LIN {X 0,Y 271.494,Z 602.071,A -85,B 0,C 180,E1 12019.317,E2 12019.317} C_VEL
LIN {X 0,Y 274.769,Z 581.052,A -85,B 0,C 180,E1 12017.936,E2 12017.936} C_VEL
LIN {X 0,Y 277.472,Z 558.924,A -85,B 0,C 180,E1 12016.896,E2 12016.896} C_VEL
LIN {X 0,Y 292.736,Z 402.476,A -85,B 0,C 180,E1 12011.469,E2 12011.469} C_VEL
LIN {X 0,Y 280.402,Z 378.491,A -85,B 0,C 180,E1 12008.156,E2 12008.156} C_VEL
LIN {X 0,Y 268.661,Z 357.396,A -85,B 0,C 180,E1 12004.711,E2 12004.711} C_VEL
LIN {X 0,Y 263.05,Z 347.539,A -85,B 0,C 180,E1 12002.855,E2 12002.855} C_VEL
LIN {X 0,Y 263.382,Z 346.943,A -85,B 0,C 180,E1 12002.565,E2 12002.565} C_VEL
LIN {X 0,Y 264.367,Z 347.015,A -85,B 0,C 180,E1 12002.274,E2 12002.274} C_VEL
LIN {X 0,Y 270.486,Z 361.582,A -85,B 0,C 180,E1 11998.605,E2 11998.605} C_VEL
LIN {X 0,Y 276.098,Z 377.318,A -85,B 0,C 180,E1 11995.128,E2 11995.128} C_VEL
LIN {X 0,Y 279.437,Z 389.009,A -85,B 0,C 180,E1 11992.846,E2 11992.846} C_VEL
LIN {X 0,Y 273.666,Z 431.774,A -85,B 0,C 180,E1 11987.985,E2 11987.985} C_VEL
LIN {X 0,Y 267.938,Z 475.725,A -85,B 0,C 180,E1 11982.94,E2 11982.94} C_VEL
LIN {X 0,Y 266.869,Z 485.441,A -85,B 0,C 180,E1 11981.853,E2 11981.853} C_VEL
LIN {X 0,Y 268.737,Z 511.468,A -85,B 0,C 180,E1 11980.723,E2 11980.723} C_VEL
LIN {X 0,Y 263.4,Z 629.84,A -85,B 0,C 180,E1 11977.527,E2 11977.527} C_VEL
LIN {X 0,Y 262.031,Z 646.203,A -85,B 0,C 180,E1 11976.686,E2 11976.686} C_VEL
LIN {X 0,Y 260.134,Z 661.581,A -85,B 0,C 180,E1 11975.516,E2 11975.516} C_VEL
LIN {X 0,Y 257.767,Z 676.09,A -85,B 0,C 180,E1 11974.006,E2 11974.006} C_VEL
LIN {X 0,Y 254.908,Z 690.584,A -85,B 0,C 180,E1 11972.025,E2 11972.025} C_VEL
LIN {X 0,Y 251.971,Z 703.426,A -85,B 0,C 180,E1 11969.752,E2 11969.752} C_VEL
LIN {X 0,Y 248.964,Z 715.561,A -85,B 0,C 180,E1 11967.01,E2 11967.01} C_VEL
LIN {X 0,Y 246.29,Z 725.681,A -85,B 0,C 180,E1 11964.066,E2 11964.066} C_VEL
LIN {X 0,Y 243.991,Z 734.43,A -85,B 0,C 180,E1 11960.806,E2 11960.806} C_VEL
LIN {X 0,Y 242.244,Z 741.402,A -85,B 0,C 180,E1 11957.367,E2 11957.367} C_VEL
LIN {X 0,Y 241.046,Z 746.913,A -85,B 0,C 180,E1 11953.619,E2 11953.619} C_VEL
LIN {X 0,Y 240.46,Z 750.406,A -85,B 0,C 180,E1 11950.01,E2 11950.01} C_VEL
LIN {X 0,Y 240.251,Z 752.346,A -85,B 0,C 180,E1 11946.194,E2 11946.194} C_VEL
LIN {X 0,Y 240.321,Z 752.618,A -85,B 0,C 180,E1 11942.401,E2 11942.401} C_VEL
LIN {X 0,Y 240.756,Z 751.048,A -85,B 0,C 180,E1 11938.451,E2 11938.451} C_VEL
LIN {X 0,Y 241.757,Z 747.721,A -85,B 0,C 180,E1 11934.565,E2 11934.565} C_VEL
LIN {X 0,Y 243.459,Z 742.459,A -85,B 0,C 180,E1 11930.772,E2 11930.772} C_VEL
LIN {X 0,Y 245.836,Z 735.559,A -85,B 0,C 180,E1 11927.222,E2 11927.222} C_VEL
LIN {X 0,Y 248.868,Z 726.664,A -85,B 0,C 180,E1 11923.842,E2 11923.842} C_VEL
LIN {X 0,Y 251.845,Z 717.662,A -85,B 0,C 180,E1 11921.176,E2 11921.176} C_VEL
LIN {X 0,Y 252.569,Z 712.778,A -85,B 0,C 180,E1 11919.813,E2 11919.813} C_VEL
LIN {X 0,Y 251.472,Z 702.77,A -85,B 0,C 180,E1 11917.085,E2 11917.085} C_VEL
LIN {X 0,Y 251.596,Z 696.374,A -85,B 0,C 180,E1 11915.677,E2 11915.677} C_VEL
LIN {X 0,Y 252.14,Z 693.786,A -85,B 0,C 180,E1 11915.218,E2 11915.218} C_VEL
LIN {X 0,Y 255.515,Z 680.254,A -85,B 0,C 180,E1 11913.284,E2 11913.284} C_VEL
LIN {X 0,Y 258.516,Z 665.707,A -85,B 0,C 180,E1 11911.697,E2 11911.697} C_VEL
LIN {X 0,Y 260.934,Z 650.294,A -85,B 0,C 180,E1 11910.46,E2 11910.46} C_VEL
LIN {X 0,Y 262.727,Z 633.392,A -85,B 0,C 180,E1 11909.54,E2 11909.54} C_VEL
LIN {X 0,Y 264.426,Z 602.955,A -85,B 0,C 180,E1 11908.631,E2 11908.631} C_VEL
LIN {X 0,Y 269.357,Z 511.316,A -85,B 0,C 180,E1 11906.141,E2 11906.141} C_VEL
LIN {X 0,Y 267.623,Z 486.252,A -85,B 0,C 180,E1 11904.737,E2 11904.737} C_VEL
LIN {X 0,Y 274.663,Z 440.447,A -85,B 0,C 180,E1 11899.475,E2 11899.475} C_VEL
LIN {X 0,Y 281.678,Z 396.905,A -85,B 0,C 180,E1 11894.519,E2 11894.519} C_VEL
LIN {X 0,Y 278.503,Z 384.661,A -85,B 0,C 180,E1 11891.599,E2 11891.599} C_VEL
LIN {X 0,Y 275.112,Z 374.138,A -85,B 0,C 180,E1 11888.57,E2 11888.57} C_VEL
LIN {X 0,Y 271.329,Z 364.565,A -85,B 0,C 180,E1 11885.287,E2 11885.287} C_VEL
LIN {X 0,Y 268.101,Z 357.243,A -85,B 0,C 180,E1 11882.138,E2 11882.138} C_VEL
LIN {X 0,Y 265.809,Z 352.672,A -85,B 0,C 180,E1 11879.785,E2 11879.785} C_VEL
LIN {X 0,Y 264.137,Z 348.957,A -85,B 0,C 180,E1 11877.614,E2 11877.614} C_VEL
LIN {X 0,Y 262.032,Z 344.964,A -85,B 0,C 180,E1 11874.746,E2 11874.746} C_VEL
LIN {X 0,Y 261.21,Z 343.736,A -85,B 0,C 180,E1 11873.407,E2 11873.407} C_VEL
LIN {X 0,Y 259.249,Z 339.266,A -85,B 0,C 180,E1 11868.395,E2 11868.395} C_VEL
LIN {X 0,Y 258.446,Z 338.509,A -85,B 0,C 180,E1 11862.437,E2 11862.437} C_VEL
LIN {X 0,Y 259.489,Z 339.421,A -85,B 0,C 180,E1 11858.053,E2 11858.053} C_VEL
LIN {X 0,Y 259.379,Z 345.514,A -85,B 0,C 180,E1 11855.155,E2 11855.155} C_VEL
LIN {X 0,Y 259.573,Z 350.003,A -85,B 0,C 180,E1 11853.615,E2 11853.615} C_VEL
LIN {X 0,Y 271.338,Z 369.415,A -85,B 0,C 180,E1 11849.925,E2 11849.925} C_VEL
LIN {X 0,Y 283.805,Z 391.256,A -85,B 0,C 180,E1 11846.389,E2 11846.389} C_VEL
LIN {X 0,Y 291.694,Z 406.109,A -85,B 0,C 180,E1 11844.305,E2 11844.305} C_VEL
LIN {X 0,Y 274.876,Z 575.506,A -85,B 0,C 180,E1 11838.587,E2 11838.587} C_VEL
LIN {X 0,Y 271.832,Z 596.932,A -85,B 0,C 180,E1 11837.513,E2 11837.513} C_VEL
LIN {X 0,Y 268.025,Z 618.404,A -85,B 0,C 180,E1 11836.049,E2 11836.049} C_VEL
LIN {X 0,Y 263.729,Z 638.906,A -85,B 0,C 180,E1 11834.23,E2 11834.23} C_VEL
LIN {X 0,Y 259.299,Z 657.672,A -85,B 0,C 180,E1 11832.136,E2 11832.136} C_VEL
LIN {X 0,Y 254.654,Z 675.677,A -85,B 0,C 180,E1 11829.656,E2 11829.656} C_VEL
LIN {X 0,Y 249.995,Z 692.7,A -85,B 0,C 180,E1 11826.779,E2 11826.779} C_VEL
LIN {X 0,Y 245.488,Z 708.606,A -85,B 0,C 180,E1 11823.493,E2 11823.493} C_VEL
LIN {X 0,Y 241.388,Z 723.196,A -85,B 0,C 180,E1 11819.802,E2 11819.802} C_VEL
LIN {X 0,Y 238.102,Z 736.125,A -85,B 0,C 180,E1 11816.021,E2 11816.021} C_VEL
LIN {X 0,Y 235.984,Z 746.974,A -85,B 0,C 180,E1 11812.676,E2 11812.676} C_VEL
LIN {X 0,Y 234.301,Z 755.943,A -85,B 0,C 180,E1 11809.18,E2 11809.18} C_VEL
LIN {X 0,Y 233.077,Z 763.404,A -85,B 0,C 180,E1 11805.422,E2 11805.422} C_VEL
LIN {X 0,Y 232.378,Z 769.258,A -85,B 0,C 180,E1 11801.413,E2 11801.413} C_VEL
LIN {X 0,Y 232.172,Z 772.992,A -85,B 0,C 180,E1 11797.669,E2 11797.669} C_VEL
LIN {X 0,Y 232.21,Z 775.067,A -85,B 0,C 180,E1 11793.948,E2 11793.948} C_VEL
LIN {X 0,Y 232.292,Z 775.579,A -85,B 0,C 180,E1 11790.244,E2 11790.244} C_VEL
LIN {X 0,Y 232.233,Z 775.277,A -85,B 0,C 180,E1 11787.036,E2 11787.036} C_VEL
LIN {X 0,Y 232.091,Z 774.894,A -85,B 0,C 180,E1 11782.82,E2 11782.82} C_VEL
LIN {X 0,Y 232.348,Z 773.008,A -85,B 0,C 180,E1 11778.077,E2 11778.077} C_VEL
LIN {X 0,Y 233.577,Z 769.389,A -85,B 0,C 180,E1 11773.075,E2 11773.075} C_VEL
LIN {X 0,Y 236.446,Z 763.468,A -85,B 0,C 180,E1 11767.628,E2 11767.628} C_VEL
LIN {X 0,Y 241.157,Z 755.58,A -85,B 0,C 180,E1 11762.329,E2 11762.329} C_VEL
LIN {X 0,Y 248.196,Z 745.291,A -85,B 0,C 180,E1 11757.051,E2 11757.051} C_VEL
LIN {X 0,Y 257.447,Z 732.968,A -85,B 0,C 180,E1 11752.145,E2 11752.145} C_VEL
LIN {X 0,Y 269.502,Z 718.104,A -85,B 0,C 180,E1 11747.526,E2 11747.526} C_VEL
LIN {X 0,Y 283.352,Z 702.222,A -85,B 0,C 180,E1 11743.663,E2 11743.663} C_VEL
LIN {X 0,Y 289.035,Z 696.015,A -85,B 0,C 180,E1 11742.353,E2 11742.353} C_VEL
LIN {X 0,Y 275.346,Z 709.401,A -85,B 0,C 180,E1 11738.917,E2 11738.917} C_VEL
LIN {X 0,Y 263.037,Z 721.802,A -85,B 0,C 180,E1 11734.762,E2 11734.762} C_VEL
LIN {X 0,Y 252.946,Z 732.321,A -85,B 0,C 180,E1 11730.132,E2 11730.132} C_VEL
LIN {X 0,Y 245.312,Z 740.47,A -85,B 0,C 180,E1 11725.338,E2 11725.338} C_VEL
LIN {X 0,Y 239.818,Z 746.395,A -85,B 0,C 180,E1 11720.5,E2 11720.5} C_VEL
LIN {X 0,Y 236.002,Z 750.456,A -85,B 0,C 180,E1 11715.48,E2 11715.48} C_VEL
LIN {X 0,Y 233.765,Z 752.545,A -85,B 0,C 180,E1 11710.597,E2 11710.597} C_VEL
LIN {X 0,Y 232.675,Z 752.869,A -85,B 0,C 180,E1 11705.919,E2 11705.919} C_VEL
LIN {X 0,Y 232.274,Z 751.624,A -85,B 0,C 180,E1 11701.479,E2 11701.479} C_VEL
LIN {X 0,Y 232.176,Z 749.013,A -85,B 0,C 180,E1 11697.284,E2 11697.284} C_VEL
LIN {X 0,Y 232.325,Z 744.909,A -85,B 0,C 180,E1 11693.078,E2 11693.078} C_VEL
LIN {X 0,Y 232.887,Z 739.168,A -85,B 0,C 180,E1 11688.859,E2 11688.859} C_VEL
LIN {X 0,Y 234.051,Z 731.644,A -85,B 0,C 180,E1 11684.64,E2 11684.64} C_VEL
LIN {X 0,Y 235.982,Z 722.115,A -85,B 0,C 180,E1 11680.443,E2 11680.443} C_VEL
LIN {X 0,Y 238.593,Z 711.091,A -85,B 0,C 180,E1 11676.539,E2 11676.539} C_VEL
LIN {X 0,Y 241.789,Z 698.652,A -85,B 0,C 180,E1 11672.942,E2 11672.942} C_VEL
LIN {X 0,Y 245.586,Z 684.276,A -85,B 0,C 180,E1 11669.543,E2 11669.543} C_VEL
LIN {X 0,Y 249.754,Z 668.328,A -85,B 0,C 180,E1 11666.463,E2 11666.463} C_VEL
LIN {X 0,Y 254.158,Z 650.692,A -85,B 0,C 180,E1 11663.695,E2 11663.695} C_VEL
LIN {X 0,Y 258.477,Z 632.032,A -85,B 0,C 180,E1 11661.337,E2 11661.337} C_VEL
LIN {X 0,Y 262.541,Z 612.369,A -85,B 0,C 180,E1 11659.364,E2 11659.364} C_VEL
LIN {X 0,Y 266.041,Z 592.568,A -85,B 0,C 180,E1 11657.821,E2 11657.821} C_VEL
LIN {X 0,Y 269.162,Z 571.164,A -85,B 0,C 180,E1 11656.579,E2 11656.579} C_VEL
LIN {X 0,Y 272.248,Z 542.164,A -85,B 0,C 180,E1 11655.408,E2 11655.408} C_VEL
LIN {X 0,Y 286.213,Z 405.215,A -85,B 0,C 180,E1 11650.561,E2 11650.561} C_VEL
LIN {X 0,Y 274.152,Z 381.732,A -85,B 0,C 180,E1 11647.196,E2 11647.196} C_VEL
LIN {X 0,Y 263.313,Z 362.162,A -85,B 0,C 180,E1 11643.9,E2 11643.9} C_VEL
LIN {X 0,Y 259.462,Z 355.12,A -85,B 0,C 180,E1 11642.544,E2 11642.544} C_VEL
LIN {X 0,Y 259.948,Z 354.608,A -85,B 0,C 180,E1 11642.197,E2 11642.197} C_VEL
LIN {X 0,Y 265.947,Z 369.757,A -85,B 0,C 180,E1 11638.386,E2 11638.386} C_VEL
LIN {X 0,Y 270.932,Z 384.639,A -85,B 0,C 180,E1 11635.115,E2 11635.115} C_VEL
LIN {X 0,Y 272.965,Z 392.002,A -85,B 0,C 180,E1 11633.66,E2 11633.66} C_VEL
LIN {X 0,Y 267.1,Z 433.334,A -85,B 0,C 180,E1 11628.895,E2 11628.895} C_VEL
LIN {X 0,Y 261.43,Z 474.987,A -85,B 0,C 180,E1 11624.058,E2 11624.058} C_VEL
LIN {X 0,Y 260.198,Z 485.826,A -85,B 0,C 180,E1 11622.836,E2 11622.836} C_VEL
LIN {X 0,Y 262.029,Z 512.287,A -85,B 0,C 180,E1 11621.656,E2 11621.656} C_VEL
LIN {X 0,Y 256.451,Z 630.322,A -85,B 0,C 180,E1 11618.395,E2 11618.395} C_VEL
LIN {X 0,Y 255.011,Z 646.741,A -85,B 0,C 180,E1 11617.529,E2 11617.529} C_VEL
LIN {X 0,Y 253.07,Z 661.849,A -85,B 0,C 180,E1 11616.354,E2 11616.354} C_VEL
LIN {X 0,Y 250.605,Z 676.391,A -85,B 0,C 180,E1 11614.809,E2 11614.809} C_VEL
LIN {X 0,Y 247.624,Z 690.905,A -85,B 0,C 180,E1 11612.78,E2 11612.78} C_VEL
LIN {X 0,Y 244.589,Z 703.65,A -85,B 0,C 180,E1 11610.471,E2 11610.471} C_VEL
LIN {X 0,Y 241.413,Z 715.913,A -85,B 0,C 180,E1 11607.629,E2 11607.629} C_VEL
LIN {X 0,Y 238.505,Z 726.419,A -85,B 0,C 180,E1 11604.47,E2 11604.47} C_VEL
LIN {X 0,Y 236.196,Z 734.801,A -85,B 0,C 180,E1 11601.237,E2 11601.237} C_VEL
LIN {X 0,Y 234.356,Z 741.78,A -85,B 0,C 180,E1 11597.686,E2 11597.686} C_VEL
LIN {X 0,Y 233.093,Z 747.297,A -85,B 0,C 180,E1 11593.813,E2 11593.813} C_VEL
LIN {X 0,Y 232.482,Z 750.755,A -85,B 0,C 180,E1 11590.141,E2 11590.141} C_VEL
LIN {X 0,Y 232.258,Z 752.739,A -85,B 0,C 180,E1 11586.133,E2 11586.133} C_VEL
LIN {X 0,Y 232.336,Z 753.025,A -85,B 0,C 180,E1 11582.308,E2 11582.308} C_VEL
LIN {X 0,Y 232.802,Z 751.526,A -85,B 0,C 180,E1 11578.256,E2 11578.256} C_VEL
LIN {X 0,Y 233.903,Z 748.174,A -85,B 0,C 180,E1 11574.156,E2 11574.156} C_VEL
LIN {X 0,Y 235.607,Z 743.314,A -85,B 0,C 180,E1 11570.468,E2 11570.468} C_VEL
LIN {X 0,Y 238.092,Z 736.561,A -85,B 0,C 180,E1 11566.807,E2 11566.807} C_VEL
LIN {X 0,Y 241.11,Z 728.302,A -85,B 0,C 180,E1 11563.477,E2 11563.477} C_VEL
LIN {X 0,Y 244.661,Z 718.184,A -85,B 0,C 180,E1 11560.353,E2 11560.353} C_VEL
LIN {X 0,Y 248.154,Z 707.442,A -85,B 0,C 180,E1 11557.767,E2 11557.767} C_VEL
LIN {X 0,Y 251.913,Z 694.598,A -85,B 0,C 180,E1 11555.355,E2 11555.355} C_VEL
LIN {X 0,Y 252.14,Z 693.786,A -85,B 0,C 180,E1 11555.218,E2 11555.218} C_VEL
LIN {X 0,Y 252.943,Z 687.681,A -85,B 0,C 180,E1 11554.142,E2 11554.142} C_VEL
LIN {X 0,Y 251.846,Z 673.719,A -85,B 0,C 180,E1 11551.616,E2 11551.616} C_VEL
LIN {X 0,Y 252.061,Z 667.063,A -85,B 0,C 180,E1 11550.711,E2 11550.711} C_VEL
LIN {X 0,Y 252.375,Z 665.07,A -85,B 0,C 180,E1 11550.503,E2 11550.503} C_VEL
LIN {X 0,Y 254.891,Z 649.347,A -85,B 0,C 180,E1 11549.257,E2 11549.257} C_VEL
LIN {X 0,Y 256.677,Z 632.86,A -85,B 0,C 180,E1 11548.369,E2 11548.369} C_VEL
LIN {X 0,Y 260.151,Z 572.276,A -85,B 0,C 180,E1 11546.628,E2 11546.628} C_VEL
LIN {X 0,Y 263.538,Z 512.271,A -85,B 0,C 180,E1 11544.968,E2 11544.968} C_VEL
LIN {X 0,Y 261.859,Z 487.034,A -85,B 0,C 180,E1 11543.517,E2 11543.517} C_VEL
LIN {X 0,Y 269.118,Z 441.982,A -85,B 0,C 180,E1 11538.298,E2 11538.298} C_VEL
LIN {X 0,Y 276.117,Z 400.724,A -85,B 0,C 180,E1 11533.561,E2 11533.561} C_VEL
LIN {X 0,Y 273.39,Z 389.42,A -85,B 0,C 180,E1 11530.751,E2 11530.751} C_VEL
LIN {X 0,Y 270.594,Z 380.2,A -85,B 0,C 180,E1 11528.02,E2 11528.02} C_VEL
LIN {X 0,Y 267.148,Z 370.865,A -85,B 0,C 180,E1 11524.724,E2 11524.724} C_VEL
LIN {X 0,Y 264.039,Z 363.618,A -85,B 0,C 180,E1 11521.52,E2 11521.52} C_VEL
LIN {X 0,Y 262.156,Z 359.505,A -85,B 0,C 180,E1 11519.345,E2 11519.345} C_VEL
LIN {X 0,Y 260.523,Z 355.857,A -85,B 0,C 180,E1 11517.141,E2 11517.141} C_VEL
LIN {X 0,Y 258.425,Z 351.439,A -85,B 0,C 180,E1 11513.782,E2 11513.782} C_VEL
LIN {X 0,Y 256.516,Z 347.354,A -85,B 0,C 180,E1 11509.173,E2 11509.173} C_VEL
LIN {X 0,Y 256.252,Z 346.625,A -85,B 0,C 180,E1 11507.837,E2 11507.837} C_VEL
LIN {X 0,Y 255.772,Z 346.054,A -85,B 0,C 180,E1 11502.248,E2 11502.248} C_VEL
LIN {X 0,Y 256.678,Z 346.655,A -85,B 0,C 180,E1 11498.521,E2 11498.521} C_VEL
LIN {X 0,Y 256.428,Z 352.391,A -85,B 0,C 180,E1 11495.833,E2 11495.833} C_VEL
LIN {X 0,Y 256.52,Z 358.28,A -85,B 0,C 180,E1 11493.775,E2 11493.775} C_VEL
LIN {X 0,Y 268.181,Z 377.95,A -85,B 0,C 180,E1 11490.059,E2 11490.059} C_VEL
LIN {X 0,Y 280.331,Z 399.558,A -85,B 0,C 180,E1 11486.573,E2 11486.573} C_VEL
LIN {X 0,Y 285.231,Z 409.114,A -85,B 0,C 180,E1 11485.228,E2 11485.228} C_VEL
LIN {X 0,Y 268.013,Z 575.619,A -85,B 0,C 180,E1 11479.454,E2 11479.454} C_VEL
LIN {X 0,Y 264.884,Z 596.863,A -85,B 0,C 180,E1 11478.36,E2 11478.36} C_VEL
LIN {X 0,Y 260.978,Z 618.204,A -85,B 0,C 180,E1 11476.869,E2 11476.869} C_VEL
LIN {X 0,Y 256.566,Z 638.64,A -85,B 0,C 180,E1 11475.013,E2 11475.013} C_VEL
LIN {X 0,Y 251.791,Z 658.206,A -85,B 0,C 180,E1 11472.765,E2 11472.765} C_VEL
LIN {X 0,Y 247.008,Z 676.133,A -85,B 0,C 180,E1 11470.209,E2 11470.209} C_VEL
LIN {X 0,Y 242.353,Z 692.634,A -85,B 0,C 180,E1 11467.331,E2 11467.331} C_VEL
LIN {X 0,Y 237.684,Z 708.623,A -85,B 0,C 180,E1 11463.918,E2 11463.918} C_VEL
LIN {X 0,Y 233.255,Z 724.496,A -85,B 0,C 180,E1 11459.889,E2 11459.889} C_VEL
LIN {X 0,Y 230.681,Z 736.731,A -85,B 0,C 180,E1 11456.764,E2 11456.764} C_VEL
LIN {X 0,Y 228.298,Z 747.641,A -85,B 0,C 180,E1 11453.211,E2 11453.211} C_VEL
LIN {X 0,Y 226.476,Z 756.403,A -85,B 0,C 180,E1 11449.601,E2 11449.601} C_VEL
LIN {X 0,Y 225.149,Z 763.621,A -85,B 0,C 180,E1 11445.714,E2 11445.714} C_VEL
LIN {X 0,Y 224.392,Z 769.313,A -85,B 0,C 180,E1 11441.564,E2 11441.564} C_VEL
LIN {X 0,Y 224.168,Z 773.013,A -85,B 0,C 180,E1 11437.429,E2 11437.429} C_VEL
LIN {X 0,Y 224.224,Z 774.858,A -85,B 0,C 180,E1 11433.576,E2 11433.576} C_VEL
LIN {X 0,Y 224.304,Z 775.142,A -85,B 0,C 180,E1 11429.742,E2 11429.742} C_VEL
LIN {X 0,Y 224.239,Z 774.681,A -85,B 0,C 180,E1 11426.674,E2 11426.674} C_VEL
LIN {X 0,Y 224.104,Z 774.334,A -85,B 0,C 180,E1 11422.047,E2 11422.047} C_VEL
LIN {X 0,Y 224.526,Z 772.338,A -85,B 0,C 180,E1 11416.87,E2 11416.87} C_VEL
LIN {X 0,Y 226.218,Z 768.472,A -85,B 0,C 180,E1 11411.441,E2 11411.441} C_VEL
LIN {X 0,Y 229.7,Z 762.535,A -85,B 0,C 180,E1 11405.845,E2 11405.845} C_VEL
LIN {X 0,Y 235.455,Z 754.321,A -85,B 0,C 180,E1 11400.206,E2 11400.206} C_VEL
LIN {X 0,Y 243.487,Z 744.149,A -85,B 0,C 180,E1 11394.905,E2 11394.905} C_VEL
LIN {X 0,Y 254.295,Z 731.59,A -85,B 0,C 180,E1 11389.845,E2 11389.845} C_VEL
LIN {X 0,Y 267.584,Z 717.288,A -85,B 0,C 180,E1 11385.371,E2 11385.371} C_VEL
LIN {X 0,Y 279.674,Z 705.089,A -85,B 0,C 180,E1 11382.299,E2 11382.299} C_VEL
LIN {X 0,Y 265.174,Z 717.754,A -85,B 0,C 180,E1 11378.472,E2 11378.472} C_VEL
LIN {X 0,Y 252.612,Z 729.11,A -85,B 0,C 180,E1 11373.923,E2 11373.923} C_VEL
LIN {X 0,Y 242.853,Z 738.169,A -85,B 0,C 180,E1 11369.066,E2 11369.066} C_VEL
LIN {X 0,Y 235.58,Z 744.978,A -85,B 0,C 180,E1 11364.044,E2 11364.044} C_VEL
LIN {X 0,Y 230.269,Z 749.837,A -85,B 0,C 180,E1 11358.742,E2 11358.742} C_VEL
LIN {X 0,Y 226.95,Z 752.62,A -85,B 0,C 180,E1 11353.502,E2 11353.502} C_VEL
LIN {X 0,Y 225.16,Z 753.534,A -85,B 0,C 180,E1 11348.426,E2 11348.426} C_VEL
LIN {X 0,Y 224.408,Z 752.743,A -85,B 0,C 180,E1 11343.553,E2 11343.553} C_VEL
LIN {X 0,Y 224.198,Z 750.439,A -85,B 0,C 180,E1 11338.977,E2 11338.977} C_VEL
LIN {X 0,Y 224.234,Z 746.715,A -85,B 0,C 180,E1 11334.626,E2 11334.626} C_VEL
LIN {X 0,Y 224.634,Z 741.414,A -85,B 0,C 180,E1 11330.261,E2 11330.261} C_VEL
LIN {X 0,Y 225.605,Z 734.39,A -85,B 0,C 180,E1 11325.891,E2 11325.891} C_VEL
LIN {X 0,Y 227.332,Z 725.447,A -85,B 0,C 180,E1 11321.537,E2 11321.537} C_VEL
LIN {X 0,Y 229.76,Z 715.051,A -85,B 0,C 180,E1 11317.482,E2 11317.482} C_VEL
LIN {X 0,Y 232.803,Z 703.296,A -85,B 0,C 180,E1 11313.744,E2 11313.744} C_VEL
LIN {X 0,Y 236.612,Z 689.242,A -85,B 0,C 180,E1 11310.089,E2 11310.089} C_VEL
LIN {X 0,Y 240.871,Z 673.589,A -85,B 0,C 180,E1 11306.773,E2 11306.773} C_VEL
LIN {X 0,Y 245.425,Z 656.201,A -85,B 0,C 180,E1 11303.79,E2 11303.79} C_VEL
LIN {X 0,Y 249.925,Z 637.749,A -85,B 0,C 180,E1 11301.251,E2 11301.251} C_VEL
LIN {X 0,Y 254.246,Z 618.089,A -85,B 0,C 180,E1 11299.095,E2 11299.095} C_VEL
LIN {X 0,Y 258.195,Z 597.49,A -85,B 0,C 180,E1 11297.336,E2 11297.336} C_VEL
LIN {X 0,Y 261.59,Z 576.13,A -85,B 0,C 180,E1 11295.958,E2 11295.958} C_VEL
LIN {X 0,Y 264.306,Z 553.841,A -85,B 0,C 180,E1 11294.945,E2 11294.945} C_VEL
LIN {X 0,Y 279.796,Z 408.146,A -85,B 0,C 180,E1 11289.649,E2 11289.649} C_VEL
LIN {X 0,Y 267.51,Z 384.104,A -85,B 0,C 180,E1 11286.066,E2 11286.066} C_VEL
LIN {X 0,Y 256.178,Z 363.663,A -85,B 0,C 180,E1 11282.459,E2 11282.459} C_VEL
LIN {X 0,Y 255.776,Z 362.628,A -85,B 0,C 180,E1 11282.119,E2 11282.119} C_VEL
LIN {X 0,Y 256.512,Z 364.958,A -85,B 0,C 180,E1 11281.388,E2 11281.388} C_VEL
LIN {X 0,Y 262.035,Z 379.972,A -85,B 0,C 180,E1 11277.715,E2 11277.715} C_VEL
LIN {X 0,Y 266.545,Z 394.897,A -85,B 0,C 180,E1 11274.52,E2 11274.52} C_VEL
LIN {X 0,Y 260.248,Z 437.782,A -85,B 0,C 180,E1 11269.529,E2 11269.529} C_VEL
LIN {X 0,Y 254.152,Z 480.628,A -85,B 0,C 180,E1 11264.469,E2 11264.469} C_VEL
LIN {X 0,Y 253.586,Z 486.33,A -85,B 0,C 180,E1 11263.854,E2 11263.854} C_VEL
LIN {X 0,Y 255.345,Z 513.166,A -85,B 0,C 180,E1 11262.622,E2 11262.622} C_VEL
LIN {X 0,Y 249.556,Z 630.626,A -85,B 0,C 180,E1 11259.312,E2 11259.312} C_VEL
LIN {X 0,Y 248.068,Z 646.977,A -85,B 0,C 180,E1 11258.433,E2 11258.433} C_VEL
LIN {X 0,Y 246.058,Z 662.048,A -85,B 0,C 180,E1 11257.239,E2 11257.239} C_VEL
LIN {X 0,Y 243.492,Z 676.649,A -85,B 0,C 180,E1 11255.658,E2 11255.658} C_VEL
LIN {X 0,Y 240.384,Z 691.194,A -85,B 0,C 180,E1 11253.58,E2 11253.58} C_VEL
LIN {X 0,Y 237.215,Z 703.971,A -85,B 0,C 180,E1 11251.21,E2 11251.21} C_VEL
LIN {X 0,Y 233.891,Z 716.252,A -85,B 0,C 180,E1 11248.288,E2 11248.288} C_VEL
LIN {X 0,Y 231.057,Z 726.056,A -85,B 0,C 180,E1 11245.287,E2 11245.287} C_VEL
LIN {X 0,Y 228.39,Z 735.262,A -85,B 0,C 180,E1 11241.657,E2 11241.657} C_VEL
LIN {X 0,Y 226.476,Z 742.158,A -85,B 0,C 180,E1 11238.027,E2 11238.027} C_VEL
LIN {X 0,Y 225.141,Z 747.679,A -85,B 0,C 180,E1 11234.021,E2 11234.021} C_VEL
LIN {X 0,Y 224.477,Z 751.264,A -85,B 0,C 180,E1 11230.027,E2 11230.027} C_VEL
LIN {X 0,Y 224.265,Z 753.211,A -85,B 0,C 180,E1 11225.788,E2 11225.788} C_VEL
LIN {X 0,Y 224.38,Z 753.375,A -85,B 0,C 180,E1 11221.817,E2 11221.817} C_VEL
LIN {X 0,Y 224.933,Z 751.769,A -85,B 0,C 180,E1 11217.629,E2 11217.629} C_VEL
LIN {X 0,Y 226.112,Z 748.514,A -85,B 0,C 180,E1 11213.593,E2 11213.593} C_VEL
LIN {X 0,Y 228.106,Z 743.271,A -85,B 0,C 180,E1 11209.558,E2 11209.558} C_VEL
LIN {X 0,Y 230.839,Z 736.383,A -85,B 0,C 180,E1 11205.789,E2 11205.789} C_VEL
LIN {X 0,Y 234.113,Z 727.94,A -85,B 0,C 180,E1 11202.371,E2 11202.371} C_VEL
LIN {X 0,Y 237.761,Z 718.16,A -85,B 0,C 180,E1 11199.311,E2 11199.311} C_VEL
LIN {X 0,Y 241.601,Z 706.878,A -85,B 0,C 180,E1 11196.581,E2 11196.581} C_VEL
LIN {X 0,Y 245.637,Z 693.669,A -85,B 0,C 180,E1 11194.098,E2 11194.098} C_VEL
LIN {X 0,Y 249.157,Z 680.091,A -85,B 0,C 180,E1 11192.147,E2 11192.147} C_VEL
LIN {X 0,Y 252.375,Z 665.07,A -85,B 0,C 180,E1 11190.503,E2 11190.503} C_VEL
LIN {X 0,Y 252.892,Z 658.091,A -85,B 0,C 180,E1 11189.73,E2 11189.73} C_VEL
LIN {X 0,Y 251.256,Z 644.385,A -85,B 0,C 180,E1 11188.045,E2 11188.045} C_VEL
LIN {X 0,Y 250.603,Z 636.11,A -85,B 0,C 180,E1 11187.324,E2 11187.324} C_VEL
LIN {X 0,Y 250.705,Z 632.868,A -85,B 0,C 180,E1 11187.162,E2 11187.162} C_VEL
LIN {X 0,Y 257.896,Z 513.32,A -85,B 0,C 180,E1 11183.734,E2 11183.734} C_VEL
LIN {X 0,Y 256.313,Z 487.239,A -85,B 0,C 180,E1 11182.175,E2 11182.175} C_VEL
LIN {X 0,Y 264.093,Z 441.625,A -85,B 0,C 180,E1 11176.837,E2 11176.837} C_VEL
LIN {X 0,Y 270.737,Z 404.278,A -85,B 0,C 180,E1 11172.478,E2 11172.478} C_VEL
LIN {X 0,Y 268.321,Z 393.587,A -85,B 0,C 180,E1 11169.654,E2 11169.654} C_VEL
LIN {X 0,Y 265.327,Z 384.015,A -85,B 0,C 180,E1 11166.709,E2 11166.709} C_VEL
LIN {X 0,Y 262.014,Z 374.57,A -85,B 0,C 180,E1 11163.063,E2 11163.063} C_VEL
LIN {X 0,Y 258.867,Z 366.992,A -85,B 0,C 180,E1 11159.337,E2 11159.337} C_VEL
LIN {X 0,Y 256.999,Z 362.781,A -85,B 0,C 180,E1 11156.655,E2 11156.655} C_VEL
LIN {X 0,Y 255.254,Z 358.691,A -85,B 0,C 180,E1 11153.478,E2 11153.478} C_VEL
LIN {X 0,Y 253.568,Z 354.666,A -85,B 0,C 180,E1 11148.86,E2 11148.86} C_VEL
LIN {X 0,Y 253.229,Z 353.955,A -85,B 0,C 180,E1 11147.215,E2 11147.215} C_VEL
LIN {X 0,Y 253.131,Z 353.618,A -85,B 0,C 180,E1 11141.58,E2 11141.58} C_VEL
LIN {X 0,Y 253.853,Z 354.345,A -85,B 0,C 180,E1 11138.755,E2 11138.755} C_VEL
LIN {X 0,Y 253.469,Z 359.89,A -85,B 0,C 180,E1 11136.275,E2 11136.275} C_VEL
LIN {X 0,Y 253.446,Z 366.618,A -85,B 0,C 180,E1 11133.936,E2 11133.936} C_VEL
LIN {X 0,Y 265.525,Z 387.341,A -85,B 0,C 180,E1 11130.04,E2 11130.04} C_VEL
LIN {X 0,Y 278.506,Z 411.075,A -85,B 0,C 180,E1 11126.282,E2 11126.282} C_VEL
LIN {X 0,Y 278.766,Z 412.273,A -85,B 0,C 180,E1 11126.173,E2 11126.173} C_VEL
LIN {X 0,Y 261.181,Z 575.534,A -85,B 0,C 180,E1 11120.356,E2 11120.356} C_VEL
LIN {X 0,Y 257.863,Z 597.286,A -85,B 0,C 180,E1 11119.203,E2 11119.203} C_VEL
LIN {X 0,Y 253.989,Z 617.808,A -85,B 0,C 180,E1 11117.734,E2 11117.734} C_VEL
LIN {X 0,Y 249.454,Z 638.208,A -85,B 0,C 180,E1 11115.841,E2 11115.841} C_VEL
LIN {X 0,Y 244.562,Z 657.679,A -85,B 0,C 180,E1 11113.554,E2 11113.554} C_VEL
LIN {X 0,Y 239.614,Z 675.697,A -85,B 0,C 180,E1 11110.925,E2 11110.925} C_VEL
LIN {X 0,Y 234.634,Z 692.797,A -85,B 0,C 180,E1 11107.849,E2 11107.849} C_VEL
LIN {X 0,Y 229.682,Z 709.307,A -85,B 0,C 180,E1 11104.198,E2 11104.198} C_VEL
LIN {X 0,Y 226.058,Z 725.598,A -85,B 0,C 180,E1 11100.717,E2 11100.717} C_VEL
LIN {X 0,Y 223.452,Z 736.747,A -85,B 0,C 180,E1 11097.73,E2 11097.73} C_VEL
LIN {X 0,Y 220.803,Z 747.635,A -85,B 0,C 180,E1 11094.047,E2 11094.047} C_VEL
LIN {X 0,Y 218.785,Z 756.288,A -85,B 0,C 180,E1 11090.32,E2 11090.32} C_VEL
LIN {X 0,Y 217.227,Z 763.841,A -85,B 0,C 180,E1 11086.029,E2 11086.029} C_VEL
LIN {X 0,Y 216.438,Z 769.056,A -85,B 0,C 180,E1 11081.995,E2 11081.995} C_VEL
LIN {X 0,Y 216.175,Z 772.697,A -85,B 0,C 180,E1 11077.705,E2 11077.705} C_VEL
LIN {X 0,Y 216.227,Z 774.497,A -85,B 0,C 180,E1 11073.709,E2 11073.709} C_VEL
LIN {X 0,Y 216.314,Z 774.74,A -85,B 0,C 180,E1 11069.732,E2 11069.732} C_VEL
LIN {X 0,Y 216.248,Z 774.064,A -85,B 0,C 180,E1 11066.286,E2 11066.286} C_VEL
LIN {X 0,Y 216.12,Z 773.83,A -85,B 0,C 180,E1 11061.484,E2 11061.484} C_VEL
LIN {X 0,Y 216.608,Z 772.136,A -85,B 0,C 180,E1 11056.381,E2 11056.381} C_VEL
LIN {X 0,Y 218.617,Z 768.29,A -85,B 0,C 180,E1 11050.493,E2 11050.493} C_VEL
LIN {X 0,Y 222.507,Z 762.588,A -85,B 0,C 180,E1 11044.727,E2 11044.727} C_VEL
LIN {X 0,Y 228.901,Z 754.64,A -85,B 0,C 180,E1 11038.885,E2 11038.885} C_VEL
LIN {X 0,Y 237.898,Z 744.644,A -85,B 0,C 180,E1 11033.355,E2 11033.355} C_VEL
LIN {X 0,Y 249.536,Z 732.752,A -85,B 0,C 180,E1 11028.304,E2 11028.304} C_VEL
LIN {X 0,Y 264.301,Z 718.748,A -85,B 0,C 180,E1 11023.731,E2 11023.731} C_VEL
LIN {X 0,Y 270.243,Z 713.321,A -85,B 0,C 180,E1 11022.269,E2 11022.269} C_VEL
LIN {X 0,Y 254.966,Z 725.279,A -85,B 0,C 180,E1 11018.001,E2 11018.001} C_VEL
LIN {X 0,Y 242.522,Z 735.299,A -85,B 0,C 180,E1 11013.18,E2 11013.18} C_VEL
LIN {X 0,Y 233.128,Z 742.927,A -85,B 0,C 180,E1 11008.149,E2 11008.149} C_VEL
LIN {X 0,Y 226.145,Z 748.507,A -85,B 0,C 180,E1 11002.896,E2 11002.896} C_VEL
LIN {X 0,Y 221.197,Z 752.221,A -85,B 0,C 180,E1 10997.357,E2 10997.357} C_VEL
LIN {X 0,Y 218.355,Z 753.923,A -85,B 0,C 180,E1 10992.159,E2 10992.159} C_VEL
LIN {X 0,Y 216.847,Z 753.922,A -85,B 0,C 180,E1 10986.884,E2 10986.884} C_VEL
LIN {X 0,Y 216.309,Z 752.398,A -85,B 0,C 180,E1 10982.118,E2 10982.118} C_VEL
LIN {X 0,Y 216.179,Z 749.422,A -85,B 0,C 180,E1 10977.527,E2 10977.527} C_VEL
LIN {X 0,Y 216.321,Z 745.098,A -85,B 0,C 180,E1 10973.097,E2 10973.097} C_VEL
LIN {X 0,Y 216.981,Z 738.666,A -85,B 0,C 180,E1 10968.301,E2 10968.301} C_VEL
LIN {X 0,Y 218.301,Z 730.723,A -85,B 0,C 180,E1 10963.775,E2 10963.775} C_VEL
LIN {X 0,Y 220.483,Z 720.753,A -85,B 0,C 180,E1 10959.284,E2 10959.284} C_VEL
LIN {X 0,Y 223.414,Z 709.249,A -85,B 0,C 180,E1 10955.121,E2 10955.121} C_VEL
LIN {X 0,Y 227.1,Z 695.837,A -85,B 0,C 180,E1 10951.185,E2 10951.185} C_VEL
LIN {X 0,Y 231.34,Z 680.776,A -85,B 0,C 180,E1 10947.592,E2 10947.592} C_VEL
LIN {X 0,Y 235.948,Z 664.01,A -85,B 0,C 180,E1 10944.36,E2 10944.36} C_VEL
LIN {X 0,Y 240.593,Z 646.172,A -85,B 0,C 180,E1 10941.588,E2 10941.588} C_VEL
LIN {X 0,Y 245.292,Z 626.405,A -85,B 0,C 180,E1 10939.137,E2 10939.137} C_VEL
LIN {X 0,Y 249.469,Z 606.611,A -85,B 0,C 180,E1 10937.206,E2 10937.206} C_VEL
LIN {X 0,Y 253.18,Z 585.962,A -85,B 0,C 180,E1 10935.651,E2 10935.651} C_VEL
LIN {X 0,Y 256.316,Z 564.259,A -85,B 0,C 180,E1 10934.459,E2 10934.459} C_VEL
LIN {X 0,Y 273.266,Z 410.887,A -85,B 0,C 180,E1 10928.667,E2 10928.667} C_VEL
LIN {X 0,Y 262.067,Z 388.774,A -85,B 0,C 180,E1 10925.28,E2 10925.28} C_VEL
LIN {X 0,Y 252.395,Z 371.07,A -85,B 0,C 180,E1 10922.098,E2 10922.098} C_VEL
LIN {X 0,Y 251.628,Z 371.456,A -85,B 0,C 180,E1 10921.674,E2 10921.674} C_VEL
LIN {X 0,Y 256.638,Z 386.082,A -85,B 0,C 180,E1 10918.002,E2 10918.002} C_VEL
LIN {X 0,Y 260.149,Z 397.891,A -85,B 0,C 180,E1 10915.416,E2 10915.416} C_VEL
LIN {X 0,Y 253.926,Z 438.358,A -85,B 0,C 180,E1 10910.637,E2 10910.637} C_VEL
LIN {X 0,Y 247.536,Z 481.768,A -85,B 0,C 180,E1 10905.464,E2 10905.464} C_VEL
LIN {X 0,Y 247.05,Z 486.725,A -85,B 0,C 180,E1 10904.932,E2 10904.932} C_VEL
LIN {X 0,Y 248.738,Z 513.972,A -85,B 0,C 180,E1 10903.64,E2 10903.64} C_VEL
LIN {X 0,Y 242.7,Z 631.12,A -85,B 0,C 180,E1 10900.266,E2 10900.266} C_VEL
LIN {X 0,Y 241.14,Z 647.499,A -85,B 0,C 180,E1 10899.363,E2 10899.363} C_VEL
LIN {X 0,Y 238.914,Z 663.402,A -85,B 0,C 180,E1 10898.062,E2 10898.062} C_VEL
LIN {X 0,Y 236.059,Z 678.632,A -85,B 0,C 180,E1 10896.325,E2 10896.325} C_VEL
LIN {X 0,Y 232.846,Z 692.861,A -85,B 0,C 180,E1 10894.189,E2 10894.189} C_VEL
LIN {X 0,Y 229.366,Z 706.104,A -85,B 0,C 180,E1 10891.588,E2 10891.588} C_VEL
LIN {X 0,Y 226.131,Z 717.449,A -85,B 0,C 180,E1 10888.736,E2 10888.736} C_VEL
LIN {X 0,Y 222.981,Z 727.817,A -85,B 0,C 180,E1 10885.373,E2 10885.373} C_VEL
LIN {X 0,Y 220.478,Z 736.081,A -85,B 0,C 180,E1 10881.921,E2 10881.921} C_VEL
LIN {X 0,Y 218.37,Z 743.358,A -85,B 0,C 180,E1 10877.844,E2 10877.844} C_VEL
LIN {X 0,Y 217.125,Z 748.36,A -85,B 0,C 180,E1 10873.964,E2 10873.964} C_VEL
LIN {X 0,Y 216.449,Z 751.904,A -85,B 0,C 180,E1 10869.677,E2 10869.677} C_VEL
LIN {X 0,Y 216.272,Z 753.681,A -85,B 0,C 180,E1 10865.416,E2 10865.416} C_VEL
LIN {X 0,Y 216.431,Z 753.708,A -85,B 0,C 180,E1 10861.289,E2 10861.289} C_VEL
LIN {X 0,Y 217.129,Z 751.913,A -85,B 0,C 180,E1 10856.775,E2 10856.775} C_VEL
LIN {X 0,Y 218.538,Z 748.345,A -85,B 0,C 180,E1 10852.523,E2 10852.523} C_VEL
LIN {X 0,Y 220.87,Z 742.794,A -85,B 0,C 180,E1 10848.287,E2 10848.287} C_VEL
LIN {X 0,Y 223.81,Z 735.833,A -85,B 0,C 180,E1 10844.54,E2 10844.54} C_VEL
LIN {X 0,Y 227.565,Z 726.772,A -85,B 0,C 180,E1 10840.896,E2 10840.896} C_VEL
LIN {X 0,Y 231.512,Z 716.57,A -85,B 0,C 180,E1 10837.788,E2 10837.788} C_VEL
LIN {X 0,Y 235.837,Z 704.394,A -85,B 0,C 180,E1 10834.915,E2 10834.915} C_VEL
LIN {X 0,Y 239.957,Z 691.059,A -85,B 0,C 180,E1 10832.516,E2 10832.516} C_VEL
LIN {X 0,Y 243.641,Z 677.153,A -85,B 0,C 180,E1 10830.59,E2 10830.59} C_VEL
LIN {X 0,Y 246.772,Z 662.268,A -85,B 0,C 180,E1 10829.05,E2 10829.05} C_VEL
LIN {X 0,Y 249.31,Z 646.142,A -85,B 0,C 180,E1 10827.839,E2 10827.839} C_VEL
LIN {X 0,Y 250.705,Z 632.868,A -85,B 0,C 180,E1 10827.162,E2 10827.162} C_VEL
LIN {X 0,Y 250.508,Z 625.322,A -85,B 0,C 180,E1 10826.738,E2 10826.738} C_VEL
LIN {X 0,Y 247.178,Z 605.499,A -85,B 0,C 180,E1 10825.161,E2 10825.161} C_VEL
LIN {X 0,Y 247.044,Z 598.979,A -85,B 0,C 180,E1 10824.857,E2 10824.857} C_VEL
LIN {X 0,Y 252.379,Z 514.396,A -85,B 0,C 180,E1 10822.447,E2 10822.447} C_VEL
LIN {X 0,Y 250.911,Z 487.444,A -85,B 0,C 180,E1 10820.773,E2 10820.773} C_VEL
LIN {X 0,Y 258.854,Z 443.464,A -85,B 0,C 180,E1 10815.573,E2 10815.573} C_VEL
LIN {X 0,Y 265.455,Z 408.125,A -85,B 0,C 180,E1 10811.406,E2 10811.406} C_VEL
LIN {X 0,Y 263.242,Z 397.681,A -85,B 0,C 180,E1 10808.52,E2 10808.52} C_VEL
LIN {X 0,Y 260.693,Z 389.136,A -85,B 0,C 180,E1 10805.724,E2 10805.724} C_VEL
LIN {X 0,Y 257.967,Z 380.891,A -85,B 0,C 180,E1 10802.444,E2 10802.444} C_VEL
LIN {X 0,Y 255.306,Z 373.868,A -85,B 0,C 180,E1 10798.879,E2 10798.879} C_VEL
LIN {X 0,Y 253.468,Z 369.676,A -85,B 0,C 180,E1 10796.156,E2 10796.156} C_VEL
LIN {X 0,Y 252.046,Z 365.92,A -85,B 0,C 180,E1 10793.166,E2 10793.166} C_VEL
LIN {X 0,Y 250.652,Z 361.942,A -85,B 0,C 180,E1 10788.496,E2 10788.496} C_VEL
LIN {X 0,Y 250.057,Z 361.041,A -85,B 0,C 180,E1 10784.223,E2 10784.223} C_VEL
LIN {X 0,Y 251.049,Z 361.654,A -85,B 0,C 180,E1 10779.24,E2 10779.24} C_VEL
LIN {X 0,Y 250.59,Z 366.24,A -85,B 0,C 180,E1 10777.167,E2 10777.167} C_VEL
LIN {X 0,Y 250.315,Z 374.957,A -85,B 0,C 180,E1 10774.095,E2 10774.095} C_VEL
LIN {X 0,Y 262.393,Z 396.063,A -85,B 0,C 180,E1 10770.149,E2 10770.149} C_VEL
LIN {X 0,Y 272.396,Z 414.775,A -85,B 0,C 180,E1 10767.171,E2 10767.171} C_VEL
LIN {X 0,Y 254.432,Z 575.008,A -85,B 0,C 180,E1 10761.31,E2 10761.31} C_VEL
LIN {X 0,Y 251.039,Z 596.637,A -85,B 0,C 180,E1 10760.141,E2 10760.141} C_VEL
LIN {X 0,Y 246.795,Z 618.373,A -85,B 0,C 180,E1 10758.543,E2 10758.543} C_VEL
LIN {X 0,Y 242.147,Z 638.593,A -85,B 0,C 180,E1 10756.608,E2 10756.608} C_VEL
LIN {X 0,Y 237.085,Z 658.088,A -85,B 0,C 180,E1 10754.243,E2 10754.243} C_VEL
LIN {X 0,Y 231.842,Z 676.526,A -85,B 0,C 180,E1 10751.448,E2 10751.448} C_VEL
LIN {X 0,Y 226.791,Z 693.347,A -85,B 0,C 180,E1 10748.303,E2 10748.303} C_VEL
LIN {X 0,Y 224.95,Z 699.747,A -85,B 0,C 180,E1 10747.029,E2 10747.029} C_VEL
LIN {X 0,Y 222.22,Z 712.919,A -85,B 0,C 180,E1 10744.689,E2 10744.689} C_VEL
LIN {X 0,Y 219.129,Z 725.901,A -85,B 0,C 180,E1 10741.8,E2 10741.8} C_VEL
LIN {X 0,Y 216.268,Z 736.876,A -85,B 0,C 180,E1 10738.735,E2 10738.735} C_VEL
LIN {X 0,Y 213.368,Z 747.654,A -85,B 0,C 180,E1 10734.941,E2 10734.941} C_VEL
LIN {X 0,Y 211.132,Z 756.177,A -85,B 0,C 180,E1 10731.091,E2 10731.091} C_VEL
LIN {X 0,Y 209.394,Z 763.67,A -85,B 0,C 180,E1 10726.645,E2 10726.645} C_VEL
LIN {X 0,Y 208.494,Z 768.795,A -85,B 0,C 180,E1 10722.459,E2 10722.459} C_VEL
LIN {X 0,Y 208.185,Z 772.382,A -85,B 0,C 180,E1 10718.003,E2 10718.003} C_VEL
LIN {X 0,Y 208.229,Z 774.139,A -85,B 0,C 180,E1 10713.852,E2 10713.852} C_VEL
LIN {X 0,Y 208.33,Z 774.357,A -85,B 0,C 180,E1 10709.997,E2 10709.997} C_VEL
LIN {X 0,Y 208.255,Z 773.413,A -85,B 0,C 180,E1 10705.867,E2 10705.867} C_VEL
LIN {X 0,Y 208.138,Z 773.329,A -85,B 0,C 180,E1 10700.876,E2 10700.876} C_VEL
LIN {X 0,Y 208.839,Z 771.599,A -85,B 0,C 180,E1 10695.263,E2 10695.263} C_VEL
LIN {X 0,Y 211.226,Z 767.895,A -85,B 0,C 180,E1 10689.203,E2 10689.203} C_VEL
LIN {X 0,Y 215.656,Z 762.405,A -85,B 0,C 180,E1 10683.271,E2 10683.271} C_VEL
LIN {X 0,Y 222.999,Z 754.531,A -85,B 0,C 180,E1 10677.141,E2 10677.141} C_VEL
LIN {X 0,Y 233.47,Z 744.408,A -85,B 0,C 180,E1 10671.296,E2 10671.296} C_VEL
LIN {X 0,Y 246.738,Z 732.553,A -85,B 0,C 180,E1 10666.134,E2 10666.134} C_VEL
LIN {X 0,Y 260.577,Z 720.951,A -85,B 0,C 180,E1 10662.181,E2 10662.181} C_VEL
LIN {X 0,Y 245.831,Z 731.225,A -85,B 0,C 180,E1 10657.89,E2 10657.89} C_VEL
LIN {X 0,Y 233.535,Z 739.915,A -85,B 0,C 180,E1 10652.938,E2 10652.938} C_VEL
LIN {X 0,Y 223.739,Z 746.776,A -85,B 0,C 180,E1 10647.405,E2 10647.405} C_VEL
LIN {X 0,Y 216.732,Z 751.437,A -85,B 0,C 180,E1 10641.657,E2 10641.657} C_VEL
LIN {X 0,Y 212.347,Z 753.972,A -85,B 0,C 180,E1 10636.128,E2 10636.128} C_VEL
LIN {X 0,Y 209.814,Z 754.763,A -85,B 0,C 180,E1 10630.71,E2 10630.71} C_VEL
LIN {X 0,Y 208.627,Z 753.948,A -85,B 0,C 180,E1 10625.499,E2 10625.499} C_VEL
LIN {X 0,Y 208.24,Z 751.631,A -85,B 0,C 180,E1 10620.549,E2 10620.549} C_VEL
LIN {X 0,Y 208.192,Z 747.984,A -85,B 0,C 180,E1 10615.868,E2 10615.868} C_VEL
LIN {X 0,Y 208.52,Z 742.631,A -85,B 0,C 180,E1 10611.046,E2 10611.046} C_VEL
LIN {X 0,Y 209.469,Z 735.428,A -85,B 0,C 180,E1 10606.191,E2 10606.191} C_VEL
LIN {X 0,Y 211.218,Z 726.507,A -85,B 0,C 180,E1 10601.507,E2 10601.507} C_VEL
LIN {X 0,Y 213.734,Z 716.142,A -85,B 0,C 180,E1 10597.151,E2 10597.151} C_VEL
LIN {X 0,Y 217.162,Z 703.568,A -85,B 0,C 180,E1 10592.881,E2 10592.881} C_VEL
LIN {X 0,Y 221.23,Z 689.419,A -85,B 0,C 180,E1 10588.986,E2 10588.986} C_VEL
LIN {X 0,Y 225.803,Z 673.604,A -85,B 0,C 180,E1 10585.452,E2 10585.452} C_VEL
LIN {X 0,Y 230.439,Z 656.926,A -85,B 0,C 180,E1 10582.437,E2 10582.437} C_VEL
LIN {X 0,Y 235.234,Z 638.439,A -85,B 0,C 180,E1 10579.752,E2 10579.752} C_VEL
LIN {X 0,Y 239.786,Z 619.029,A -85,B 0,C 180,E1 10577.505,E2 10577.505} C_VEL
LIN {X 0,Y 244.082,Z 598.091,A -85,B 0,C 180,E1 10575.615,E2 10575.615} C_VEL
LIN {X 0,Y 247.764,Z 576.507,A -85,B 0,C 180,E1 10574.145,E2 10574.145} C_VEL
LIN {X 0,Y 250.691,Z 554.253,A -85,B 0,C 180,E1 10573.076,E2 10573.076} C_VEL
LIN {X 0,Y 266.856,Z 413.714,A -85,B 0,C 180,E1 10567.675,E2 10567.675} C_VEL
LIN {X 0,Y 255.082,Z 390.415,A -85,B 0,C 180,E1 10563.959,E2 10563.959} C_VEL
LIN {X 0,Y 249.203,Z 379.769,A -85,B 0,C 180,E1 10561.982,E2 10561.982} C_VEL
LIN {X 0,Y 247.528,Z 379.986,A -85,B 0,C 180,E1 10561.457,E2 10561.457} C_VEL
LIN {X 0,Y 247.772,Z 381.516,A -85,B 0,C 180,E1 10560.936,E2 10560.936} C_VEL
LIN {X 0,Y 252.534,Z 396.462,A -85,B 0,C 180,E1 10557.343,E2 10557.343} C_VEL
LIN {X 0,Y 253.805,Z 401.186,A -85,B 0,C 180,E1 10556.31,E2 10556.31} C_VEL
LIN {X 0,Y 247.15,Z 442.761,A -85,B 0,C 180,E1 10551.355,E2 10551.355} C_VEL
LIN {X 0,Y 240.542,Z 486.564,A -85,B 0,C 180,E1 10546.088,E2 10546.088} C_VEL
LIN {X 0,Y 242.209,Z 514.736,A -85,B 0,C 180,E1 10544.713,E2 10544.713} C_VEL
LIN {X 0,Y 235.918,Z 631.475,A -85,B 0,C 180,E1 10541.279,E2 10541.279} C_VEL
LIN {X 0,Y 234.284,Z 647.929,A -85,B 0,C 180,E1 10540.352,E2 10540.352} C_VEL
LIN {X 0,Y 232.019,Z 663.507,A -85,B 0,C 180,E1 10539.052,E2 10539.052} C_VEL
LIN {X 0,Y 229.18,Z 678.184,A -85,B 0,C 180,E1 10537.36,E2 10537.36} C_VEL
LIN {X 0,Y 225.917,Z 692.2,A -85,B 0,C 180,E1 10535.241,E2 10535.241} C_VEL
LIN {X 0,Y 222.426,Z 705.074,A -85,B 0,C 180,E1 10532.708,E2 10532.708} C_VEL
LIN {X 0,Y 218.942,Z 716.84,A -85,B 0,C 180,E1 10529.741,E2 10529.741} C_VEL
LIN {X 0,Y 215.822,Z 726.693,A -85,B 0,C 180,E1 10526.55,E2 10526.55} C_VEL
LIN {X 0,Y 212.897,Z 735.839,A -85,B 0,C 180,E1 10522.718,E2 10522.718} C_VEL
LIN {X 0,Y 210.739,Z 742.863,A -85,B 0,C 180,E1 10518.786,E2 10518.786} C_VEL
LIN {X 0,Y 209.246,Z 748.409,A -85,B 0,C 180,E1 10514.482,E2 10514.482} C_VEL
LIN {X 0,Y 208.528,Z 751.898,A -85,B 0,C 180,E1 10510.392,E2 10510.392} C_VEL
LIN {X 0,Y 208.282,Z 753.907,A -85,B 0,C 180,E1 10505.922,E2 10505.922} C_VEL
LIN {X 0,Y 208.413,Z 754.218,A -85,B 0,C 180,E1 10501.648,E2 10501.648} C_VEL
LIN {X 0,Y 209.021,Z 752.836,A -85,B 0,C 180,E1 10497.284,E2 10497.284} C_VEL
LIN {X 0,Y 210.373,Z 749.7,A -85,B 0,C 180,E1 10492.876,E2 10492.876} C_VEL
LIN {X 0,Y 212.475,Z 745.045,A -85,B 0,C 180,E1 10488.796,E2 10488.796} C_VEL
LIN {X 0,Y 215.469,Z 738.451,A -85,B 0,C 180,E1 10484.772,E2 10484.772} C_VEL
LIN {X 0,Y 219.129,Z 730.303,A -85,B 0,C 180,E1 10481.077,E2 10481.077} C_VEL
LIN {X 0,Y 223.412,Z 720.13,A -85,B 0,C 180,E1 10477.619,E2 10477.619} C_VEL
LIN {X 0,Y 227.614,Z 709.314,A -85,B 0,C 180,E1 10474.776,E2 10474.776} C_VEL
LIN {X 0,Y 232.077,Z 696.286,A -85,B 0,C 180,E1 10472.151,E2 10472.151} C_VEL
LIN {X 0,Y 235.875,Z 683.505,A -85,B 0,C 180,E1 10470.153,E2 10470.153} C_VEL
LIN {X 0,Y 239.411,Z 669.014,A -85,B 0,C 180,E1 10468.432,E2 10468.432} C_VEL
LIN {X 0,Y 242.242,Z 654.163,A -85,B 0,C 180,E1 10467.114,E2 10467.114} C_VEL
LIN {X 0,Y 244.365,Z 638.259,A -85,B 0,C 180,E1 10466.136,E2 10466.136} C_VEL
LIN {X 0,Y 245.77,Z 619.713,A -85,B 0,C 180,E1 10465.45,E2 10465.45} C_VEL
LIN {X 0,Y 247.044,Z 598.979,A -85,B 0,C 180,E1 10464.857,E2 10464.857} C_VEL
LIN {X 0,Y 246.827,Z 591.391,A -85,B 0,C 180,E1 10464.477,E2 10464.477} C_VEL
LIN {X 0,Y 243.814,Z 571.542,A -85,B 0,C 180,E1 10462.851,E2 10462.851} C_VEL
LIN {X 0,Y 243.739,Z 565.021,A -85,B 0,C 180,E1 10462.533,E2 10462.533} C_VEL
LIN {X 0,Y 247.01,Z 515.369,A -85,B 0,C 180,E1 10461.094,E2 10461.094} C_VEL
LIN {X 0,Y 245.652,Z 488.238,A -85,B 0,C 180,E1 10459.362,E2 10459.362} C_VEL
LIN {X 0,Y 254.225,Z 443.085,A -85,B 0,C 180,E1 10453.987,E2 10453.987} C_VEL
LIN {X 0,Y 260.412,Z 412.111,A -85,B 0,C 180,E1 10450.285,E2 10450.285} C_VEL
LIN {X 0,Y 258.365,Z 402.518,A -85,B 0,C 180,E1 10447.562,E2 10447.562} C_VEL
LIN {X 0,Y 256.136,Z 393.747,A -85,B 0,C 180,E1 10444.479,E2 10444.479} C_VEL
LIN {X 0,Y 253.566,Z 386.286,A -85,B 0,C 180,E1 10441.357,E2 10441.357} C_VEL
LIN {X 0,Y 251.427,Z 380.065,A -85,B 0,C 180,E1 10437.95,E2 10437.95} C_VEL
LIN {X 0,Y 250.014,Z 376.591,A -85,B 0,C 180,E1 10435.643,E2 10435.643} C_VEL
LIN {X 0,Y 248.907,Z 373.157,A -85,B 0,C 180,E1 10432.812,E2 10432.812} C_VEL
LIN {X 0,Y 247.67,Z 369.022,A -85,B 0,C 180,E1 10427.646,E2 10427.646} C_VEL
LIN {X 0,Y 247.621,Z 368.632,A -85,B 0,C 180,E1 10421.886,E2 10421.886} C_VEL
LIN {X 0,Y 248.197,Z 369.164,A -85,B 0,C 180,E1 10419.607,E2 10419.607} C_VEL
LIN {X 0,Y 247.706,Z 372.966,A -85,B 0,C 180,E1 10417.952,E2 10417.952} C_VEL
LIN {X 0,Y 247.234,Z 383.401,A -85,B 0,C 180,E1 10414.232,E2 10414.232} C_VEL
LIN {X 0,Y 260.302,Z 406.834,A -85,B 0,C 180,E1 10409.917,E2 10409.917} C_VEL
LIN {X 0,Y 265.966,Z 417.879,A -85,B 0,C 180,E1 10408.177,E2 10408.177} C_VEL
LIN {X 0,Y 247.654,Z 574.88,A -85,B 0,C 180,E1 10402.28,E2 10402.28} C_VEL
LIN {X 0,Y 244.008,Z 597.232,A -85,B 0,C 180,E1 10401.03,E2 10401.03} C_VEL
LIN {X 0,Y 239.656,Z 618.703,A -85,B 0,C 180,E1 10399.399,E2 10399.399} C_VEL
LIN {X 0,Y 234.816,Z 639.044,A -85,B 0,C 180,E1 10397.389,E2 10397.389} C_VEL
LIN {X 0,Y 229.483,Z 658.904,A -85,B 0,C 180,E1 10394.893,E2 10394.893} C_VEL
LIN {X 0,Y 223.881,Z 677.931,A -85,B 0,C 180,E1 10391.883,E2 10391.883} C_VEL
LIN {X 0,Y 221.404,Z 686.158,A -85,B 0,C 180,E1 10390.39,E2 10390.39} C_VEL
LIN {X 0,Y 218.973,Z 698.995,A -85,B 0,C 180,E1 10388.551,E2 10388.551} C_VEL
LIN {X 0,Y 215.945,Z 712.149,A -85,B 0,C 180,E1 10386.177,E2 10386.177} C_VEL
LIN {X 0,Y 212.554,Z 725.18,A -85,B 0,C 180,E1 10383.227,E2 10383.227} C_VEL
LIN {X 0,Y 209.385,Z 736.197,A -85,B 0,C 180,E1 10380.089,E2 10380.089} C_VEL
LIN {X 0,Y 206.173,Z 746.992,A -85,B 0,C 180,E1 10376.184,E2 10376.184} C_VEL
LIN {X 0,Y 203.671,Z 755.576,A -85,B 0,C 180,E1 10372.207,E2 10372.207} C_VEL
LIN {X 0,Y 201.684,Z 763.092,A -85,B 0,C 180,E1 10367.599,E2 10367.599} C_VEL
LIN {X 0,Y 200.61,Z 768.274,A -85,B 0,C 180,E1 10363.251,E2 10363.251} C_VEL
LIN {X 0,Y 200.197,Z 771.94,A -85,B 0,C 180,E1 10358.555,E2 10358.555} C_VEL
LIN {X 0,Y 200.221,Z 773.706,A -85,B 0,C 180,E1 10354.293,E2 10354.293} C_VEL
LIN {X 0,Y 200.333,Z 773.971,A -85,B 0,C 180,E1 10350.283,E2 10350.283} C_VEL
LIN {X 0,Y 200.295,Z 772.826,A -85,B 0,C 180,E1 10346.276,E2 10346.276} C_VEL
LIN {X 0,Y 200.16,Z 772.82,A -85,B 0,C 180,E1 10340.509,E2 10340.509} C_VEL
LIN {X 0,Y 200.96,Z 771.316,A -85,B 0,C 180,E1 10334.707,E2 10334.707} C_VEL
LIN {X 0,Y 203.772,Z 767.741,A -85,B 0,C 180,E1 10328.102,E2 10328.102} C_VEL
LIN {X 0,Y 209.25,Z 762.034,A -85,B 0,C 180,E1 10321.453,E2 10321.453} C_VEL
LIN {X 0,Y 217.872,Z 754.105,A -85,B 0,C 180,E1 10314.992,E2 10314.992} C_VEL
LIN {X 0,Y 229.955,Z 743.969,A -85,B 0,C 180,E1 10308.959,E2 10308.959} C_VEL
LIN {X 0,Y 245.059,Z 732.211,A -85,B 0,C 180,E1 10303.763,E2 10303.763} C_VEL
LIN {X 0,Y 250.94,Z 727.824,A -85,B 0,C 180,E1 10302.136,E2 10302.136} C_VEL
LIN {X 0,Y 236.066,Z 736.975,A -85,B 0,C 180,E1 10297.582,E2 10297.582} C_VEL
LIN {X 0,Y 223.912,Z 744.431,A -85,B 0,C 180,E1 10292.401,E2 10292.401} C_VEL
LIN {X 0,Y 214.325,Z 750.091,A -85,B 0,C 180,E1 10286.605,E2 10286.605} C_VEL
LIN {X 0,Y 207.845,Z 753.565,A -85,B 0,C 180,E1 10280.853,E2 10280.853} C_VEL
LIN {X 0,Y 203.692,Z 755.226,A -85,B 0,C 180,E1 10275.079,E2 10275.079} C_VEL
LIN {X 0,Y 201.414,Z 755.191,A -85,B 0,C 180,E1 10269.428,E2 10269.428} C_VEL
LIN {X 0,Y 200.441,Z 753.513,A -85,B 0,C 180,E1 10263.889,E2 10263.889} C_VEL
LIN {X 0,Y 200.194,Z 750.466,A -85,B 0,C 180,E1 10258.854,E2 10258.854} C_VEL
LIN {X 0,Y 200.265,Z 746.046,A -85,B 0,C 180,E1 10253.981,E2 10253.981} C_VEL
LIN {X 0,Y 200.8,Z 740.01,A -85,B 0,C 180,E1 10249.092,E2 10249.092} C_VEL
LIN {X 0,Y 202.065,Z 732.181,A -85,B 0,C 180,E1 10244.207,E2 10244.207} C_VEL
LIN {X 0,Y 204.249,Z 722.337,A -85,B 0,C 180,E1 10239.361,E2 10239.361} C_VEL
LIN {X 0,Y 207.251,Z 710.975,A -85,B 0,C 180,E1 10234.877,E2 10234.877} C_VEL
LIN {X 0,Y 211.07,Z 697.754,A -85,B 0,C 180,E1 10230.653,E2 10230.653} C_VEL
LIN {X 0,Y 215.499,Z 682.9,A -85,B 0,C 180,E1 10226.804,E2 10226.804} C_VEL
LIN {X 0,Y 220.332,Z 666.479,A -85,B 0,C 180,E1 10223.362,E2 10223.362} C_VEL
LIN {X 0,Y 225.199,Z 649.082,A -85,B 0,C 180,E1 10220.421,E2 10220.421} C_VEL
LIN {X 0,Y 230.125,Z 629.881,A -85,B 0,C 180,E1 10217.833,E2 10217.833} C_VEL
LIN {X 0,Y 234.746,Z 609.704,A -85,B 0,C 180,E1 10215.69,E2 10215.69} C_VEL
LIN {X 0,Y 238.893,Z 588.471,A -85,B 0,C 180,E1 10213.953,E2 10213.953} C_VEL
LIN {X 0,Y 242.386,Z 566.63,A -85,B 0,C 180,E1 10212.643,E2 10212.643} C_VEL
LIN {X 0,Y 260.37,Z 416.349,A -85,B 0,C 180,E1 10206.634,E2 10206.634} C_VEL
LIN {X 0,Y 249.217,Z 394.288,A -85,B 0,C 180,E1 10202.967,E2 10202.967} C_VEL
LIN {X 0,Y 246.051,Z 388.346,A -85,B 0,C 180,E1 10201.863,E2 10201.863} C_VEL
LIN {X 0,Y 243.328,Z 388.829,A -85,B 0,C 180,E1 10201.149,E2 10201.149} C_VEL
LIN {X 0,Y 243.265,Z 389.649,A -85,B 0,C 180,E1 10200.791,E2 10200.791} C_VEL
LIN {X 0,Y 247.504,Z 404.236,A -85,B 0,C 180,E1 10197.281,E2 10197.281} C_VEL
LIN {X 0,Y 240.851,Z 444.3,A -85,B 0,C 180,E1 10192.455,E2 10192.455} C_VEL
LIN {X 0,Y 234.151,Z 487.041,A -85,B 0,C 180,E1 10187.267,E2 10187.267} C_VEL
LIN {X 0,Y 235.723,Z 515.556,A -85,B 0,C 180,E1 10185.829,E2 10185.829} C_VEL
LIN {X 0,Y 229.181,Z 631.841,A -85,B 0,C 180,E1 10182.338,E2 10182.338} C_VEL
LIN {X 0,Y 227.486,Z 648.235,A -85,B 0,C 180,E1 10181.396,E2 10181.396} C_VEL
LIN {X 0,Y 225.189,Z 663.46,A -85,B 0,C 180,E1 10180.104,E2 10180.104} C_VEL
LIN {X 0,Y 222.291,Z 677.993,A -85,B 0,C 180,E1 10178.409,E2 10178.409} C_VEL
LIN {X 0,Y 218.776,Z 692.523,A -85,B 0,C 180,E1 10176.168,E2 10176.168} C_VEL
LIN {X 0,Y 215.175,Z 705.27,A -85,B 0,C 180,E1 10173.599,E2 10173.599} C_VEL
LIN {X 0,Y 211.522,Z 717.075,A -85,B 0,C 180,E1 10170.545,E2 10170.545} C_VEL
LIN {X 0,Y 208.22,Z 727.044,A -85,B 0,C 180,E1 10167.222,E2 10167.222} C_VEL
LIN {X 0,Y 205.163,Z 736.141,A -85,B 0,C 180,E1 10163.286,E2 10163.286} C_VEL
LIN {X 0,Y 202.885,Z 743.192,A -85,B 0,C 180,E1 10159.21,E2 10159.21} C_VEL
LIN {X 0,Y 201.304,Z 748.755,A -85,B 0,C 180,E1 10154.741,E2 10154.741} C_VEL
LIN {X 0,Y 200.54,Z 752.289,A -85,B 0,C 180,E1 10150.449,E2 10150.449} C_VEL
LIN {X 0,Y 200.289,Z 754.29,A -85,B 0,C 180,E1 10145.84,E2 10145.84} C_VEL
LIN {X 0,Y 200.442,Z 754.618,A -85,B 0,C 180,E1 10141.392,E2 10141.392} C_VEL
LIN {X 0,Y 201.12,Z 753.254,A -85,B 0,C 180,E1 10136.852,E2 10136.852} C_VEL
LIN {X 0,Y 202.668,Z 750.003,A -85,B 0,C 180,E1 10132.127,E2 10132.127} C_VEL
LIN {X 0,Y 205.095,Z 745.048,A -85,B 0,C 180,E1 10127.724,E2 10127.724} C_VEL
LIN {X 0,Y 208.385,Z 738.359,A -85,B 0,C 180,E1 10123.576,E2 10123.576} C_VEL
LIN {X 0,Y 212.29,Z 730.165,A -85,B 0,C 180,E1 10119.834,E2 10119.834} C_VEL
LIN {X 0,Y 216.951,Z 719.717,A -85,B 0,C 180,E1 10116.249,E2 10116.249} C_VEL
LIN {X 0,Y 221.429,Z 708.663,A -85,B 0,C 180,E1 10113.353,E2 10113.353} C_VEL
LIN {X 0,Y 226.107,Z 695.641,A -85,B 0,C 180,E1 10110.724,E2 10110.724} C_VEL
LIN {X 0,Y 230.179,Z 682.341,A -85,B 0,C 180,E1 10108.67,E2 10108.67} C_VEL
LIN {X 0,Y 233.865,Z 667.618,A -85,B 0,C 180,E1 10106.95,E2 10106.95} C_VEL
LIN {X 0,Y 236.815,Z 652.159,A -85,B 0,C 180,E1 10105.627,E2 10105.627} C_VEL
LIN {X 0,Y 239.007,Z 635.151,A -85,B 0,C 180,E1 10104.644,E2 10104.644} C_VEL
LIN {X 0,Y 241.126,Z 604.367,A -85,B 0,C 180,E1 10103.663,E2 10103.663} C_VEL
LIN {X 0,Y 243.739,Z 565.021,A -85,B 0,C 180,E1 10102.533,E2 10102.533} C_VEL
LIN {X 0,Y 243.588,Z 557.436,A -85,B 0,C 180,E1 10102.141,E2 10102.141} C_VEL
LIN {X 0,Y 240.924,Z 537.596,A -85,B 0,C 180,E1 10100.456,E2 10100.456} C_VEL
LIN {X 0,Y 240.921,Z 531.076,A -85,B 0,C 180,E1 10100.135,E2 10100.135} C_VEL
LIN {X 0,Y 241.844,Z 516.339,A -85,B 0,C 180,E1 10099.668,E2 10099.668} C_VEL
LIN {X 0,Y 240.7,Z 488.445,A -85,B 0,C 180,E1 10097.809,E2 10097.809} C_VEL
LIN {X 0,Y 250.037,Z 441.986,A -85,B 0,C 180,E1 10092.237,E2 10092.237} C_VEL
LIN {X 0,Y 255.466,Z 416.113,A -85,B 0,C 180,E1 10089.121,E2 10089.121} C_VEL
LIN {X 0,Y 253.561,Z 406.795,A -85,B 0,C 180,E1 10086.34,E2 10086.34} C_VEL
LIN {X 0,Y 251.505,Z 398.358,A -85,B 0,C 180,E1 10083.191,E2 10083.191} C_VEL
LIN {X 0,Y 249.659,Z 392.262,A -85,B 0,C 180,E1 10080.46,E2 10080.46} C_VEL
LIN {X 0,Y 247.923,Z 386.935,A -85,B 0,C 180,E1 10077.458,E2 10077.458} C_VEL
LIN {X 0,Y 246.785,Z 383.748,A -85,B 0,C 180,E1 10075.29,E2 10075.29} C_VEL
LIN {X 0,Y 245.723,Z 380.287,A -85,B 0,C 180,E1 10072.284,E2 10072.284} C_VEL
LIN {X 0,Y 244.853,Z 376.48,A -85,B 0,C 180,E1 10067.395,E2 10067.395} C_VEL
LIN {X 0,Y 244.907,Z 376.153,A -85,B 0,C 180,E1 10062.171,E2 10062.171} C_VEL
LIN {X 0,Y 245.38,Z 376.711,A -85,B 0,C 180,E1 10059.985,E2 10059.985} C_VEL
LIN {X 0,Y 244.426,Z 383.414,A -85,B 0,C 180,E1 10057.387,E2 10057.387} C_VEL
LIN {X 0,Y 244.13,Z 391.988,A -85,B 0,C 180,E1 10054.364,E2 10054.364} C_VEL
LIN {X 0,Y 256.154,Z 413.953,A -85,B 0,C 180,E1 10050.315,E2 10050.315} C_VEL
LIN {X 0,Y 259.576,Z 420.766,A -85,B 0,C 180,E1 10049.222,E2 10049.222} C_VEL
LIN {X 0,Y 240.85,Z 575.105,A -85,B 0,C 180,E1 10043.268,E2 10043.268} C_VEL
LIN {X 0,Y 237.142,Z 597.038,A -85,B 0,C 180,E1 10042.007,E2 10042.007} C_VEL
LIN {X 0,Y 232.859,Z 617.623,A -85,B 0,C 180,E1 10040.416,E2 10040.416} C_VEL
LIN {X 0,Y 227.952,Z 637.756,A -85,B 0,C 180,E1 10038.4,E2 10038.4} C_VEL
LIN {X 0,Y 222.617,Z 657.151,A -85,B 0,C 180,E1 10035.936,E2 10035.936} C_VEL
LIN {X 0,Y 217.694,Z 673.964,A -85,B 0,C 180,E1 10033.361,E2 10033.361} C_VEL
LIN {X 0,Y 215.623,Z 686.451,A -85,B 0,C 180,E1 10031.888,E2 10031.888} C_VEL
LIN {X 0,Y 212.767,Z 699.832,A -85,B 0,C 180,E1 10029.896,E2 10029.896} C_VEL
LIN {X 0,Y 209.322,Z 713.417,A -85,B 0,C 180,E1 10027.342,E2 10027.342} C_VEL
LIN {X 0,Y 205.805,Z 725.58,A -85,B 0,C 180,E1 10024.467,E2 10024.467} C_VEL
LIN {X 0,Y 202.091,Z 737.226,A -85,B 0,C 180,E1 10020.963,E2 10020.963} C_VEL
LIN {X 0,Y 198.744,Z 747.446,A -85,B 0,C 180,E1 10017.07,E2 10017.07} C_VEL
LIN {X 0,Y 195.945,Z 756.03,A -85,B 0,C 180,E1 10012.814,E2 10012.814} C_VEL
LIN {X 0,Y 193.809,Z 763.358,A -85,B 0,C 180,E1 10008.028,E2 10008.028} C_VEL
LIN {X 0,Y 192.593,Z 768.562,A -85,B 0,C 180,E1 10003.201,E2 10003.201} C_VEL
LIN {X 0,Y 192.193,Z 771.943,A -85,B 0,C 180,E1 9998.372,E2 9998.372} C_VEL
LIN {X 0,Y 192.239,Z 773.475,A -85,B 0,C 180,E1 9993.874,E2 9993.874} C_VEL
LIN {X 0,Y 192.346,Z 773.473,A -85,B 0,C 180,E1 9989.699,E2 9989.699} C_VEL
LIN {X 0,Y 192.27,Z 772.058,A -85,B 0,C 180,E1 9984.925,E2 9984.925} C_VEL
LIN {X 0,Y 192.224,Z 772.198,A -85,B 0,C 180,E1 9979.507,E2 9979.507} C_VEL
LIN {X 0,Y 193.382,Z 770.706,A -85,B 0,C 180,E1 9973.166,E2 9973.166} C_VEL
LIN {X 0,Y 196.793,Z 767.238,A -85,B 0,C 180,E1 9966.332,E2 9966.332} C_VEL
LIN {X 0,Y 203.171,Z 761.676,A -85,B 0,C 180,E1 9959.452,E2 9959.452} C_VEL
LIN {X 0,Y 212.672,Z 754.195,A -85,B 0,C 180,E1 9952.999,E2 9952.999} C_VEL
LIN {X 0,Y 225.796,Z 744.608,A -85,B 0,C 180,E1 9947.002,E2 9947.002} C_VEL
LIN {X 0,Y 241.244,Z 734.039,A -85,B 0,C 180,E1 9942.105,E2 9942.105} C_VEL
LIN {X 0,Y 225.686,Z 742.38,A -85,B 0,C 180,E1 9937.05,E2 9937.05} C_VEL
LIN {X 0,Y 213.353,Z 748.778,A -85,B 0,C 180,E1 9931.344,E2 9931.344} C_VEL
LIN {X 0,Y 204.56,Z 753.017,A -85,B 0,C 180,E1 9925.475,E2 9925.475} C_VEL
LIN {X 0,Y 198.496,Z 755.406,A -85,B 0,C 180,E1 9919.417,E2 9919.417} C_VEL
LIN {X 0,Y 194.792,Z 756.034,A -85,B 0,C 180,E1 9913.354,E2 9913.354} C_VEL
LIN {X 0,Y 192.941,Z 755.001,A -85,B 0,C 180,E1 9907.443,E2 9907.443} C_VEL
LIN {X 0,Y 192.292,Z 752.428,A -85,B 0,C 180,E1 9901.787,E2 9901.787} C_VEL
LIN {X 0,Y 192.181,Z 748.624,A -85,B 0,C 180,E1 9896.718,E2 9896.718} C_VEL
LIN {X 0,Y 192.446,Z 743.289,A -85,B 0,C 180,E1 9891.634,E2 9891.634} C_VEL
LIN {X 0,Y 193.352,Z 736.135,A -85,B 0,C 180,E1 9886.464,E2 9886.464} C_VEL
LIN {X 0,Y 195.109,Z 727.288,A -85,B 0,C 180,E1 9881.459,E2 9881.459} C_VEL
LIN {X 0,Y 197.716,Z 716.934,A -85,B 0,C 180,E1 9876.767,E2 9876.767} C_VEL
LIN {X 0,Y 201.376,Z 704.175,A -85,B 0,C 180,E1 9872.108,E2 9872.108} C_VEL
LIN {X 0,Y 205.781,Z 689.734,A -85,B 0,C 180,E1 9867.859,E2 9867.859} C_VEL
LIN {X 0,Y 210.635,Z 673.908,A -85,B 0,C 180,E1 9864.108,E2 9864.108} C_VEL
LIN {X 0,Y 215.813,Z 656.319,A -85,B 0,C 180,E1 9860.771,E2 9860.771} C_VEL
LIN {X 0,Y 220.935,Z 637.705,A -85,B 0,C 180,E1 9857.948,E2 9857.948} C_VEL
LIN {X 0,Y 226.04,Z 617.124,A -85,B 0,C 180,E1 9855.483,E2 9855.483} C_VEL
LIN {X 0,Y 230.622,Z 595.825,A -85,B 0,C 180,E1 9853.521,E2 9853.521} C_VEL
LIN {X 0,Y 234.452,Z 574.128,A -85,B 0,C 180,E1 9852.038,E2 9852.038} C_VEL
LIN {X 0,Y 237.854,Z 548.874,A -85,B 0,C 180,E1 9850.816,E2 9850.816} C_VEL
LIN {X 0,Y 253.965,Z 419.148,A -85,B 0,C 180,E1 9845.572,E2 9845.572} C_VEL
LIN {X 0,Y 242.771,Z 396.87,A -85,B 0,C 180,E1 9841.713,E2 9841.713} C_VEL
LIN {X 0,Y 239.518,Z 397.687,A -85,B 0,C 180,E1 9841.008,E2 9841.008} C_VEL
LIN {X 0,Y 238.848,Z 398.328,A -85,B 0,C 180,E1 9840.539,E2 9840.539} C_VEL
LIN {X 0,Y 241.301,Z 407.722,A -85,B 0,C 180,E1 9838.265,E2 9838.265} C_VEL
LIN {X 0,Y 234.149,Z 448.676,A -85,B 0,C 180,E1 9833.268,E2 9833.268} C_VEL
LIN {X 0,Y 227.855,Z 487.355,A -85,B 0,C 180,E1 9828.52,E2 9828.52} C_VEL
LIN {X 0,Y 229.331,Z 516.378,A -85,B 0,C 180,E1 9827.007,E2 9827.007} C_VEL
LIN {X 0,Y 222.519,Z 632.315,A -85,B 0,C 180,E1 9823.457,E2 9823.457} C_VEL
LIN {X 0,Y 220.721,Z 648.894,A -85,B 0,C 180,E1 9822.478,E2 9822.478} C_VEL
LIN {X 0,Y 218.223,Z 664.643,A -85,B 0,C 180,E1 9821.098,E2 9821.098} C_VEL
LIN {X 0,Y 214.997,Z 679.863,A -85,B 0,C 180,E1 9819.236,E2 9819.236} C_VEL
LIN {X 0,Y 211.551,Z 693.391,A -85,B 0,C 180,E1 9817.061,E2 9817.061} C_VEL
LIN {X 0,Y 207.8,Z 706.031,A -85,B 0,C 180,E1 9814.418,E2 9814.418} C_VEL
LIN {X 0,Y 204.028,Z 717.672,A -85,B 0,C 180,E1 9811.298,E2 9811.298} C_VEL
LIN {X 0,Y 200.441,Z 727.963,A -85,B 0,C 180,E1 9807.716,E2 9807.716} C_VEL
LIN {X 0,Y 197.253,Z 737.027,A -85,B 0,C 180,E1 9803.601,E2 9803.601} C_VEL
LIN {X 0,Y 194.901,Z 743.942,A -85,B 0,C 180,E1 9799.361,E2 9799.361} C_VEL
LIN {X 0,Y 193.286,Z 749.42,A -85,B 0,C 180,E1 9794.707,E2 9794.707} C_VEL
LIN {X 0,Y 192.494,Z 752.984,A -85,B 0,C 180,E1 9789.955,E2 9789.955} C_VEL
LIN {X 0,Y 192.297,Z 754.839,A -85,B 0,C 180,E1 9785.096,E2 9785.096} C_VEL
LIN {X 0,Y 192.54,Z 754.923,A -85,B 0,C 180,E1 9780.444,E2 9780.444} C_VEL
LIN {X 0,Y 193.497,Z 753.171,A -85,B 0,C 180,E1 9775.365,E2 9775.365} C_VEL
LIN {X 0,Y 195.34,Z 749.675,A -85,B 0,C 180,E1 9770.617,E2 9770.617} C_VEL
LIN {X 0,Y 198.286,Z 744.167,A -85,B 0,C 180,E1 9765.909,E2 9765.909} C_VEL
LIN {X 0,Y 201.718,Z 737.65,A -85,B 0,C 180,E1 9761.974,E2 9761.974} C_VEL
LIN {X 0,Y 206.171,Z 728.807,A -85,B 0,C 180,E1 9758.019,E2 9758.019} C_VEL
LIN {X 0,Y 210.775,Z 719.016,A -85,B 0,C 180,E1 9754.699,E2 9754.699} C_VEL
LIN {X 0,Y 215.555,Z 707.71,A -85,B 0,C 180,E1 9751.766,E2 9751.766} C_VEL
LIN {X 0,Y 220.306,Z 694.992,A -85,B 0,C 180,E1 9749.215,E2 9749.215} C_VEL
LIN {X 0,Y 224.649,Z 681.173,A -85,B 0,C 180,E1 9747.115,E2 9747.115} C_VEL
LIN {X 0,Y 228.503,Z 666.193,A -85,B 0,C 180,E1 9745.394,E2 9745.394} C_VEL
LIN {X 0,Y 231.581,Z 649.983,A -85,B 0,C 180,E1 9744.063,E2 9744.063} C_VEL
LIN {X 0,Y 233.632,Z 633.879,A -85,B 0,C 180,E1 9743.173,E2 9743.173} C_VEL
LIN {X 0,Y 240.921,Z 531.076,A -85,B 0,C 180,E1 9740.135,E2 9740.135} C_VEL
LIN {X 0,Y 240.831,Z 524.601,A -85,B 0,C 180,E1 9739.783,E2 9739.783} C_VEL
LIN {X 0,Y 239.292,Z 515.474,A -85,B 0,C 180,E1 9738.843,E2 9738.843} C_VEL
LIN {X 0,Y 236.64,Z 502.462,A -85,B 0,C 180,E1 9737.283,E2 9737.283} C_VEL
LIN {X 0,Y 236.253,Z 498.21,A -85,B 0,C 180,E1 9736.916,E2 9736.916} C_VEL
LIN {X 0,Y 236.001,Z 488.293,A -85,B 0,C 180,E1 9736.151,E2 9736.151} C_VEL
LIN {X 0,Y 245.63,Z 442.94,A -85,B 0,C 180,E1 9730.674,E2 9730.674} C_VEL
LIN {X 0,Y 250.545,Z 420.117,A -85,B 0,C 180,E1 9727.915,E2 9727.915} C_VEL
LIN {X 0,Y 249.035,Z 411.206,A -85,B 0,C 180,E1 9725.068,E2 9725.068} C_VEL
LIN {X 0,Y 246.991,Z 402.953,A -85,B 0,C 180,E1 9721.857,E2 9721.857} C_VEL
LIN {X 0,Y 245.242,Z 396.209,A -85,B 0,C 180,E1 9718.365,E2 9718.365} C_VEL
LIN {X 0,Y 243.632,Z 391.048,A -85,B 0,C 180,E1 9715.057,E2 9715.057} C_VEL
LIN {X 0,Y 242.651,Z 387.553,A -85,B 0,C 180,E1 9711.947,E2 9711.947} C_VEL
LIN {X 0,Y 242.095,Z 384.318,A -85,B 0,C 180,E1 9707.841,E2 9707.841} C_VEL
LIN {X 0,Y 241.773,Z 383.578,A -85,B 0,C 180,E1 9704.407,E2 9704.407} C_VEL
LIN {X 0,Y 242.607,Z 384.034,A -85,B 0,C 180,E1 9700.5,E2 9700.5} C_VEL
LIN {X 0,Y 240.796,Z 398.417,A -85,B 0,C 180,E1 9695.205,E2 9695.205} C_VEL
LIN {X 0,Y 241.096,Z 400.768,A -85,B 0,C 180,E1 9694.451,E2 9694.451} C_VEL
LIN {X 0,Y 252.977,Z 422.935,A -85,B 0,C 180,E1 9690.394,E2 9690.394} C_VEL
LIN {X 0,Y 253.143,Z 424.148,A -85,B 0,C 180,E1 9690.284,E2 9690.284} C_VEL
LIN {X 0,Y 234.137,Z 574.847,A -85,B 0,C 180,E1 9684.317,E2 9684.317} C_VEL
LIN {X 0,Y 230.288,Z 596.905,A -85,B 0,C 180,E1 9683.018,E2 9683.018} C_VEL
LIN {X 0,Y 225.829,Z 617.631,A -85,B 0,C 180,E1 9681.372,E2 9681.372} C_VEL
LIN {X 0,Y 220.735,Z 637.855,A -85,B 0,C 180,E1 9679.288,E2 9679.288} C_VEL
LIN {X 0,Y 215.08,Z 657.785,A -85,B 0,C 180,E1 9676.675,E2 9676.675} C_VEL
LIN {X 0,Y 213.95,Z 662.473,A -85,B 0,C 180,E1 9676.12,E2 9676.12} C_VEL
LIN {X 0,Y 212.068,Z 675.752,A -85,B 0,C 180,E1 9674.814,E2 9674.814} C_VEL
LIN {X 0,Y 209.383,Z 689.628,A -85,B 0,C 180,E1 9673.063,E2 9673.063} C_VEL
LIN {X 0,Y 206.141,Z 703.112,A -85,B 0,C 180,E1 9670.9,E2 9670.9} C_VEL
LIN {X 0,Y 202.618,Z 715.323,A -85,B 0,C 180,E1 9668.441,E2 9668.441} C_VEL
LIN {X 0,Y 198.504,Z 727.958,A -85,B 0,C 180,E1 9665.217,E2 9665.217} C_VEL
LIN {X 0,Y 194.577,Z 739.128,A -85,B 0,C 180,E1 9661.606,E2 9661.606} C_VEL
LIN {X 0,Y 190.917,Z 749.082,A -85,B 0,C 180,E1 9657.439,E2 9657.439} C_VEL
LIN {X 0,Y 187.905,Z 757.538,A -85,B 0,C 180,E1 9652.853,E2 9652.853} C_VEL
LIN {X 0,Y 185.717,Z 764.291,A -85,B 0,C 180,E1 9647.867,E2 9647.867} C_VEL
LIN {X 0,Y 184.529,Z 769.111,A -85,B 0,C 180,E1 9642.832,E2 9642.832} C_VEL
LIN {X 0,Y 184.184,Z 772.034,A -85,B 0,C 180,E1 9637.796,E2 9637.796} C_VEL
LIN {X 0,Y 184.272,Z 773.191,A -85,B 0,C 180,E1 9633.107,E2 9633.107} C_VEL
LIN {X 0,Y 184.351,Z 772.849,A -85,B 0,C 180,E1 9628.754,E2 9628.754} C_VEL
LIN {X 0,Y 184.284,Z 771.346,A -85,B 0,C 180,E1 9624.392,E2 9624.392} C_VEL
LIN {X 0,Y 184.326,Z 771.567,A -85,B 0,C 180,E1 9618.419,E2 9618.419} C_VEL
LIN {X 0,Y 185.928,Z 770.111,A -85,B 0,C 180,E1 9611.498,E2 9611.498} C_VEL
LIN {X 0,Y 190.02,Z 766.792,A -85,B 0,C 180,E1 9604.436,E2 9604.436} C_VEL
LIN {X 0,Y 197.547,Z 761.296,A -85,B 0,C 180,E1 9597.206,E2 9597.206} C_VEL
LIN {X 0,Y 208.757,Z 753.751,A -85,B 0,C 180,E1 9590.427,E2 9590.427} C_VEL
LIN {X 0,Y 223.785,Z 744.252,A -85,B 0,C 180,E1 9584.364,E2 9584.364} C_VEL
LIN {X 0,Y 231.299,Z 739.685,A -85,B 0,C 180,E1 9582.027,E2 9582.027} C_VEL
LIN {X 0,Y 216.082,Z 746.688,A -85,B 0,C 180,E1 9576.817,E2 9576.817} C_VEL
LIN {X 0,Y 204.094,Z 751.883,A -85,B 0,C 180,E1 9570.956,E2 9570.956} C_VEL
LIN {X 0,Y 195.135,Z 755.238,A -85,B 0,C 180,E1 9564.521,E2 9564.521} C_VEL
LIN {X 0,Y 189.422,Z 756.643,A -85,B 0,C 180,E1 9558.144,E2 9558.144} C_VEL
LIN {X 0,Y 186.113,Z 756.324,A -85,B 0,C 180,E1 9551.779,E2 9551.779} C_VEL
LIN {X 0,Y 184.625,Z 754.377,A -85,B 0,C 180,E1 9545.593,E2 9545.593} C_VEL
LIN {X 0,Y 184.224,Z 751.132,A -85,B 0,C 180,E1 9539.999,E2 9539.999} C_VEL
LIN {X 0,Y 184.231,Z 746.534,A -85,B 0,C 180,E1 9534.705,E2 9534.705} C_VEL
LIN {X 0,Y 184.735,Z 740.339,A -85,B 0,C 180,E1 9529.395,E2 9529.395} C_VEL
LIN {X 0,Y 186.028,Z 732.351,A -85,B 0,C 180,E1 9524.09,E2 9524.09} C_VEL
LIN {X 0,Y 188.336,Z 722.351,A -85,B 0,C 180,E1 9518.837,E2 9518.837} C_VEL
LIN {X 0,Y 191.548,Z 710.819,A -85,B 0,C 180,E1 9513.992,E2 9513.992} C_VEL
LIN {X 0,Y 195.517,Z 697.858,A -85,B 0,C 180,E1 9509.582,E2 9509.582} C_VEL
LIN {X 0,Y 200.217,Z 683.004,A -85,B 0,C 180,E1 9505.49,E2 9505.49} C_VEL
LIN {X 0,Y 205.401,Z 666.436,A -85,B 0,C 180,E1 9501.813,E2 9501.813} C_VEL
LIN {X 0,Y 210.593,Z 648.943,A -85,B 0,C 180,E1 9498.703,E2 9498.703} C_VEL
LIN {X 0,Y 215.838,Z 629.725,A -85,B 0,C 180,E1 9495.982,E2 9495.982} C_VEL
LIN {X 0,Y 220.744,Z 609.527,A -85,B 0,C 180,E1 9493.741,E2 9493.741} C_VEL
LIN {X 0,Y 225.138,Z 588.374,A -85,B 0,C 180,E1 9491.935,E2 9491.935} C_VEL
LIN {X 0,Y 228.911,Z 566.276,A -85,B 0,C 180,E1 9490.546,E2 9490.546} C_VEL
LIN {X 0,Y 247.588,Z 422.026,A -85,B 0,C 180,E1 9484.469,E2 9484.469} C_VEL
LIN {X 0,Y 239.359,Z 405.458,A -85,B 0,C 180,E1 9481.551,E2 9481.551} C_VEL
LIN {X 0,Y 235.921,Z 406.764,A -85,B 0,C 180,E1 9480.854,E2 9480.854} C_VEL
LIN {X 0,Y 234.511,Z 407.098,A -85,B 0,C 180,E1 9480.35,E2 9480.35} C_VEL
LIN {X 0,Y 234.955,Z 409.752,A -85,B 0,C 180,E1 9479.583,E2 9479.583} C_VEL
LIN {X 0,Y 235.095,Z 411.255,A -85,B 0,C 180,E1 9479.284,E2 9479.284} C_VEL
LIN {X 0,Y 227.5,Z 453.154,A -85,B 0,C 180,E1 9474.128,E2 9474.128} C_VEL
LIN {X 0,Y 221.629,Z 487.647,A -85,B 0,C 180,E1 9469.831,E2 9469.831} C_VEL
LIN {X 0,Y 223.021,Z 517.149,A -85,B 0,C 180,E1 9468.246,E2 9468.246} C_VEL
LIN {X 0,Y 215.918,Z 632.684,A -85,B 0,C 180,E1 9464.635,E2 9464.635} C_VEL
LIN {X 0,Y 214.063,Z 649.126,A -85,B 0,C 180,E1 9463.646,E2 9463.646} C_VEL
LIN {X 0,Y 211.546,Z 664.466,A -85,B 0,C 180,E1 9462.283,E2 9462.283} C_VEL
LIN {X 0,Y 208.401,Z 678.939,A -85,B 0,C 180,E1 9460.508,E2 9460.508} C_VEL
LIN {X 0,Y 204.58,Z 693.449,A -85,B 0,C 180,E1 9458.151,E2 9458.151} C_VEL
LIN {X 0,Y 200.654,Z 706.168,A -85,B 0,C 180,E1 9455.436,E2 9455.436} C_VEL
LIN {X 0,Y 196.817,Z 717.49,A -85,B 0,C 180,E1 9452.332,E2 9452.332} C_VEL
LIN {X 0,Y 193.193,Z 727.477,A -85,B 0,C 180,E1 9448.817,E2 9448.817} C_VEL
LIN {X 0,Y 189.762,Z 736.705,A -85,B 0,C 180,E1 9444.561,E2 9444.561} C_VEL
LIN {X 0,Y 187.211,Z 743.822,A -85,B 0,C 180,E1 9440.163,E2 9440.163} C_VEL
LIN {X 0,Y 185.431,Z 749.427,A -85,B 0,C 180,E1 9435.323,E2 9435.323} C_VEL
LIN {X 0,Y 184.556,Z 753.097,A -85,B 0,C 180,E1 9430.509,E2 9430.509} C_VEL
LIN {X 0,Y 184.304,Z 755.053,A -85,B 0,C 180,E1 9425.654,E2 9425.654} C_VEL
LIN {X 0,Y 184.518,Z 755.416,A -85,B 0,C 180,E1 9420.744,E2 9420.744} C_VEL
LIN {X 0,Y 185.354,Z 754.108,A -85,B 0,C 180,E1 9415.879,E2 9415.879} C_VEL
LIN {X 0,Y 187.315,Z 750.745,A -85,B 0,C 180,E1 9410.57,E2 9410.57} C_VEL
LIN {X 0,Y 190.067,Z 746.008,A -85,B 0,C 180,E1 9406.026,E2 9406.026} C_VEL
LIN {X 0,Y 193.851,Z 739.381,A -85,B 0,C 180,E1 9401.598,E2 9401.598} C_VEL
LIN {X 0,Y 198.337,Z 731.178,A -85,B 0,C 180,E1 9397.59,E2 9397.59} C_VEL
LIN {X 0,Y 203.498,Z 720.941,A -85,B 0,C 180,E1 9393.871,E2 9393.871} C_VEL
LIN {X 0,Y 208.473,Z 710.061,A -85,B 0,C 180,E1 9390.858,E2 9390.858} C_VEL
LIN {X 0,Y 213.673,Z 697.07,A -85,B 0,C 180,E1 9388.115,E2 9388.115} C_VEL
LIN {X 0,Y 218.087,Z 684.209,A -85,B 0,C 180,E1 9386.034,E2 9386.034} C_VEL
LIN {X 0,Y 222.153,Z 669.622,A -85,B 0,C 180,E1 9384.255,E2 9384.255} C_VEL
LIN {X 0,Y 225.402,Z 654.619,A -85,B 0,C 180,E1 9382.9,E2 9382.9} C_VEL
LIN {X 0,Y 227.847,Z 638.126,A -85,B 0,C 180,E1 9381.884,E2 9381.884} C_VEL
LIN {X 0,Y 229.488,Z 618.665,A -85,B 0,C 180,E1 9381.173,E2 9381.173} C_VEL
LIN {X 0,Y 236.881,Z 517.514,A -85,B 0,C 180,E1 9378.186,E2 9378.186} C_VEL
LIN {X 0,Y 236.253,Z 498.21,A -85,B 0,C 180,E1 9376.916,E2 9376.916} C_VEL
LIN {X 0,Y 235.789,Z 492.147,A -85,B 0,C 180,E1 9376.266,E2 9376.266} C_VEL
LIN {X 0,Y 234.909,Z 483.19,A -85,B 0,C 180,E1 9374.657,E2 9374.657} C_VEL
LIN {X 0,Y 235.06,Z 473.605,A -85,B 0,C 180,E1 9372.749,E2 9372.749} C_VEL
LIN {X 0,Y 235.804,Z 468.863,A -85,B 0,C 180,E1 9372.052,E2 9372.052} C_VEL
LIN {X 0,Y 244.907,Z 428.771,A -85,B 0,C 180,E1 9367.245,E2 9367.245} C_VEL
LIN {X 0,Y 245.888,Z 424.258,A -85,B 0,C 180,E1 9366.656,E2 9366.656} C_VEL
LIN {X 0,Y 244.59,Z 415.72,A -85,B 0,C 180,E1 9363.751,E2 9363.751} C_VEL
LIN {X 0,Y 242.963,Z 408.393,A -85,B 0,C 180,E1 9360.708,E2 9360.708} C_VEL
LIN {X 0,Y 241.482,Z 402.215,A -85,B 0,C 180,E1 9357.39,E2 9357.39} C_VEL
LIN {X 0,Y 240.315,Z 397.785,A -85,B 0,C 180,E1 9354.27,E2 9354.27} C_VEL
LIN {X 0,Y 239.562,Z 394.77,A -85,B 0,C 180,E1 9351.535,E2 9351.535} C_VEL
LIN {X 0,Y 239.246,Z 391.417,A -85,B 0,C 180,E1 9346.958,E2 9346.958} C_VEL
LIN {X 0,Y 239.377,Z 391.156,A -85,B 0,C 180,E1 9342.75,E2 9342.75} C_VEL
LIN {X 0,Y 239.809,Z 391.49,A -85,B 0,C 180,E1 9341.022,E2 9341.022} C_VEL
LIN {X 0,Y 237.902,Z 404.084,A -85,B 0,C 180,E1 9336.37,E2 9336.37} C_VEL
LIN {X 0,Y 237.833,Z 409.265,A -85,B 0,C 180,E1 9334.609,E2 9334.609} C_VEL
LIN {X 0,Y 246.865,Z 426.525,A -85,B 0,C 180,E1 9331.421,E2 9331.421} C_VEL
LIN {X 0,Y 227.363,Z 575.096,A -85,B 0,C 180,E1 9325.376,E2 9325.376} C_VEL
LIN {X 0,Y 223.471,Z 596.678,A -85,B 0,C 180,E1 9324.074,E2 9324.074} C_VEL
LIN {X 0,Y 218.919,Z 617.233,A -85,B 0,C 180,E1 9322.406,E2 9322.406} C_VEL
LIN {X 0,Y 213.463,Z 638.211,A -85,B 0,C 180,E1 9320.185,E2 9320.185} C_VEL
LIN {X 0,Y 210.519,Z 649.065,A -85,B 0,C 180,E1 9318.88,E2 9318.88} C_VEL
LIN {X 0,Y 209.323,Z 660.622,A -85,B 0,C 180,E1 9318.032,E2 9318.032} C_VEL
LIN {X 0,Y 207.267,Z 674.027,A -85,B 0,C 180,E1 9316.749,E2 9316.749} C_VEL
LIN {X 0,Y 204.336,Z 688.148,A -85,B 0,C 180,E1 9314.992,E2 9314.992} C_VEL
LIN {X 0,Y 200.782,Z 701.77,A -85,B 0,C 180,E1 9312.819,E2 9312.819} C_VEL
LIN {X 0,Y 196.558,Z 715.349,A -85,B 0,C 180,E1 9310.047,E2 9310.047} C_VEL
LIN {X 0,Y 192.018,Z 728.138,A -85,B 0,C 180,E1 9306.69,E2 9306.69} C_VEL
LIN {X 0,Y 187.669,Z 739.331,A -85,B 0,C 180,E1 9302.913,E2 9302.913} C_VEL
LIN {X 0,Y 183.446,Z 749.807,A -85,B 0,C 180,E1 9298.302,E2 9298.302} C_VEL
LIN {X 0,Y 180.379,Z 757.492,A -85,B 0,C 180,E1 9293.852,E2 9293.852} C_VEL
LIN {X 0,Y 177.966,Z 764.139,A -85,B 0,C 180,E1 9288.674,E2 9288.674} C_VEL
LIN {X 0,Y 176.611,Z 768.858,A -85,B 0,C 180,E1 9283.418,E2 9283.418} C_VEL
LIN {X 0,Y 176.192,Z 771.712,A -85,B 0,C 180,E1 9278.152,E2 9278.152} C_VEL
LIN {X 0,Y 176.275,Z 772.814,A -85,B 0,C 180,E1 9273.248,E2 9273.248} C_VEL
LIN {X 0,Y 176.365,Z 772.479,A -85,B 0,C 180,E1 9269.022,E2 9269.022} C_VEL
LIN {X 0,Y 176.306,Z 770.772,A -85,B 0,C 180,E1 9264.464,E2 9264.464} C_VEL
LIN {X 0,Y 176.266,Z 770.679,A -85,B 0,C 180,E1 9263.054,E2 9263.054} C_VEL
LIN {X 0,Y 176.557,Z 770.88,A -85,B 0,C 180,E1 9256.571,E2 9256.571} C_VEL
LIN {X 0,Y 178.944,Z 769.314,A -85,B 0,C 180,E1 9249.043,E2 9249.043} C_VEL
LIN {X 0,Y 184.319,Z 765.832,A -85,B 0,C 180,E1 9241.483,E2 9241.483} C_VEL
LIN {X 0,Y 193.219,Z 760.434,A -85,B 0,C 180,E1 9234.212,E2 9234.212} C_VEL
LIN {X 0,Y 206.444,Z 752.847,A -85,B 0,C 180,E1 9227.305,E2 9227.305} C_VEL
LIN {X 0,Y 221.301,Z 744.666,A -85,B 0,C 180,E1 9221.964,E2 9221.964} C_VEL
LIN {X 0,Y 206.407,Z 750.458,A -85,B 0,C 180,E1 9216.57,E2 9216.57} C_VEL
LIN {X 0,Y 194.369,Z 754.651,A -85,B 0,C 180,E1 9210.272,E2 9210.272} C_VEL
LIN {X 0,Y 185.725,Z 756.942,A -85,B 0,C 180,E1 9203.476,E2 9203.476} C_VEL
LIN {X 0,Y 180.215,Z 757.341,A -85,B 0,C 180,E1 9196.436,E2 9196.436} C_VEL
LIN {X 0,Y 177.432,Z 755.995,A -85,B 0,C 180,E1 9189.732,E2 9189.732} C_VEL
LIN {X 0,Y 176.405,Z 753.242,A -85,B 0,C 180,E1 9183.573,E2 9183.573} C_VEL
LIN {X 0,Y 176.184,Z 749.377,A -85,B 0,C 180,E1 9178.047,E2 9178.047} C_VEL
LIN {X 0,Y 176.341,Z 744.31,A -85,B 0,C 180,E1 9172.833,E2 9172.833} C_VEL
LIN {X 0,Y 177.132,Z 737.32,A -85,B 0,C 180,E1 9167.281,E2 9167.281} C_VEL
LIN {X 0,Y 178.85,Z 728.436,A -85,B 0,C 180,E1 9161.755,E2 9161.755} C_VEL
LIN {X 0,Y 181.712,Z 717.415,A -85,B 0,C 180,E1 9156.316,E2 9156.316} C_VEL
LIN {X 0,Y 185.523,Z 704.794,A -85,B 0,C 180,E1 9151.336,E2 9151.336} C_VEL
LIN {X 0,Y 190.1,Z 690.615,A -85,B 0,C 180,E1 9146.837,E2 9146.837} C_VEL
LIN {X 0,Y 195.235,Z 674.865,A -85,B 0,C 180,E1 9142.819,E2 9142.819} C_VEL
LIN {X 0,Y 200.721,Z 657.439,A -85,B 0,C 180,E1 9139.264,E2 9139.264} C_VEL
LIN {X 0,Y 206.127,Z 639.078,A -85,B 0,C 180,E1 9136.286,E2 9136.286} C_VEL
LIN {X 0,Y 211.54,Z 618.674,A -85,B 0,C 180,E1 9133.682,E2 9133.682} C_VEL
LIN {X 0,Y 216.227,Z 598.503,A -85,B 0,C 180,E1 9131.685,E2 9131.685} C_VEL
LIN {X 0,Y 220.446,Z 576.842,A -85,B 0,C 180,E1 9130.057,E2 9130.057} C_VEL
LIN {X 0,Y 223.937,Z 553.777,A -85,B 0,C 180,E1 9128.83,E2 9128.83} C_VEL
LIN {X 0,Y 241.283,Z 424.9,A -85,B 0,C 180,E1 9123.341,E2 9123.341} C_VEL
LIN {X 0,Y 236.132,Z 414.398,A -85,B 0,C 180,E1 9121.461,E2 9121.461} C_VEL
LIN {X 0,Y 234.132,Z 415.034,A -85,B 0,C 180,E1 9121.044,E2 9121.044} C_VEL
LIN {X 0,Y 229.579,Z 418.365,A -85,B 0,C 180,E1 9120.203,E2 9120.203} C_VEL
LIN {X 0,Y 228.056,Z 420.524,A -85,B 0,C 180,E1 9119.7,E2 9119.7} C_VEL
LIN {X 0,Y 220.705,Z 458.49,A -85,B 0,C 180,E1 9114.921,E2 9114.921} C_VEL
LIN {X 0,Y 215.516,Z 488.142,A -85,B 0,C 180,E1 9111.199,E2 9111.199} C_VEL
LIN {X 0,Y 216.789,Z 517.936,A -85,B 0,C 180,E1 9109.546,E2 9109.546} C_VEL
LIN {X 0,Y 209.409,Z 633.039,A -85,B 0,C 180,E1 9105.884,E2 9105.884} C_VEL
LIN {X 0,Y 207.455,Z 649.632,A -85,B 0,C 180,E1 9104.865,E2 9104.865} C_VEL
LIN {X 0,Y 204.727,Z 665.469,A -85,B 0,C 180,E1 9103.417,E2 9103.417} C_VEL
LIN {X 0,Y 201.224,Z 680.683,A -85,B 0,C 180,E1 9101.467,E2 9101.467} C_VEL
LIN {X 0,Y 197.526,Z 694.032,A -85,B 0,C 180,E1 9099.214,E2 9099.214} C_VEL
LIN {X 0,Y 193.378,Z 706.849,A -85,B 0,C 180,E1 9096.386,E2 9096.386} C_VEL
LIN {X 0,Y 189.202,Z 718.602,A -85,B 0,C 180,E1 9093.033,E2 9093.033} C_VEL
LIN {X 0,Y 185.15,Z 729.144,A -85,B 0,C 180,E1 9089.075,E2 9089.075} C_VEL
LIN {X 0,Y 181.739,Z 737.915,A -85,B 0,C 180,E1 9084.755,E2 9084.755} C_VEL
LIN {X 0,Y 179.083,Z 744.968,A -85,B 0,C 180,E1 9080.037,E2 9080.037} C_VEL
LIN {X 0,Y 177.326,Z 750.379,A -85,B 0,C 180,E1 9074.971,E2 9074.971} C_VEL
LIN {X 0,Y 176.488,Z 753.875,A -85,B 0,C 180,E1 9069.787,E2 9069.787} C_VEL
LIN {X 0,Y 176.314,Z 755.598,A -85,B 0,C 180,E1 9064.834,E2 9064.834} C_VEL
LIN {X 0,Y 176.634,Z 755.745,A -85,B 0,C 180,E1 9059.753,E2 9059.753} C_VEL
LIN {X 0,Y 177.819,Z 754.039,A -85,B 0,C 180,E1 9054.217,E2 9054.217} C_VEL
LIN {X 0,Y 180.036,Z 750.598,A -85,B 0,C 180,E1 9049.053,E2 9049.053} C_VEL
LIN {X 0,Y 183.467,Z 745.165,A -85,B 0,C 180,E1 9044.003,E2 9044.003} C_VEL
LIN {X 0,Y 187.403,Z 738.745,A -85,B 0,C 180,E1 9039.806,E2 9039.806} C_VEL
LIN {X 0,Y 192.516,Z 729.865,A -85,B 0,C 180,E1 9035.571,E2 9035.571} C_VEL
LIN {X 0,Y 197.708,Z 720.11,A -85,B 0,C 180,E1 9032.075,E2 9032.075} C_VEL
LIN {X 0,Y 203.273,Z 708.331,A -85,B 0,C 180,E1 9028.898,E2 9028.898} C_VEL
LIN {X 0,Y 208.521,Z 695.65,A -85,B 0,C 180,E1 9026.285,E2 9026.285} C_VEL
LIN {X 0,Y 213.548,Z 681.105,A -85,B 0,C 180,E1 9024.039,E2 9024.039} C_VEL
LIN {X 0,Y 217.574,Z 666.676,A -85,B 0,C 180,E1 9022.374,E2 9022.374} C_VEL
LIN {X 0,Y 220.969,Z 650.243,A -85,B 0,C 180,E1 9021.016,E2 9021.016} C_VEL
LIN {X 0,Y 223.162,Z 634.229,A -85,B 0,C 180,E1 9020.134,E2 9020.134} C_VEL
LIN {X 0,Y 232.101,Z 518.594,A -85,B 0,C 180,E1 9016.632,E2 9016.632} C_VEL
LIN {X 0,Y 231.248,Z 490.16,A -85,B 0,C 180,E1 9014.64,E2 9014.64} C_VEL
LIN {X 0,Y 235.804,Z 468.863,A -85,B 0,C 180,E1 9012.052,E2 9012.052} C_VEL
LIN {X 0,Y 236.758,Z 462.355,A -85,B 0,C 180,E1 9011.05,E2 9011.05} C_VEL
LIN {X 0,Y 237.538,Z 446.235,A -85,B 0,C 180,E1 9007.699,E2 9007.699} C_VEL
LIN {X 0,Y 238.558,Z 440.651,A -85,B 0,C 180,E1 9006.854,E2 9006.854} C_VEL
LIN {X 0,Y 241.411,Z 428.499,A -85,B 0,C 180,E1 9005.348,E2 9005.348} C_VEL
LIN {X 0,Y 240.158,Z 420.19,A -85,B 0,C 180,E1 9002.372,E2 9002.372} C_VEL
LIN {X 0,Y 238.913,Z 412.936,A -85,B 0,C 180,E1 8999.042,E2 8999.042} C_VEL
LIN {X 0,Y 237.515,Z 407.242,A -85,B 0,C 180,E1 8995.655,E2 8995.655} C_VEL
LIN {X 0,Y 236.968,Z 403.964,A -85,B 0,C 180,E1 8992.972,E2 8992.972} C_VEL
LIN {X 0,Y 236.536,Z 402.082,A -85,B 0,C 180,E1 8991.248,E2 8991.248} C_VEL
LIN {X 0,Y 236.458,Z 398.899,A -85,B 0,C 180,E1 8986.802,E2 8986.802} C_VEL
LIN {X 0,Y 236.612,Z 398.663,A -85,B 0,C 180,E1 8982.737,E2 8982.737} C_VEL
LIN {X 0,Y 236.919,Z 399.079,A -85,B 0,C 180,E1 8981.548,E2 8981.548} C_VEL
LIN {X 0,Y 234.749,Z 412.233,A -85,B 0,C 180,E1 8976.665,E2 8976.665} C_VEL
LIN {X 0,Y 234.637,Z 417.994,A -85,B 0,C 180,E1 8974.728,E2 8974.728} C_VEL
LIN {X 0,Y 240.528,Z 429.545,A -85,B 0,C 180,E1 8972.574,E2 8972.574} C_VEL
LIN {X 0,Y 220.68,Z 574.974,A -85,B 0,C 180,E1 8966.5,E2 8966.5} C_VEL
LIN {X 0,Y 216.581,Z 596.883,A -85,B 0,C 180,E1 8965.138,E2 8965.138} C_VEL
LIN {X 0,Y 211.761,Z 617.854,A -85,B 0,C 180,E1 8963.381,E2 8963.381} C_VEL
LIN {X 0,Y 206.872,Z 636.815,A -85,B 0,C 180,E1 8961.417,E2 8961.417} C_VEL
LIN {X 0,Y 206.083,Z 648.541,A -85,B 0,C 180,E1 8960.764,E2 8960.764} C_VEL
LIN {X 0,Y 204.581,Z 661.318,A -85,B 0,C 180,E1 8959.826,E2 8959.826} C_VEL
LIN {X 0,Y 202.164,Z 675.307,A -85,B 0,C 180,E1 8958.439,E2 8958.439} C_VEL
LIN {X 0,Y 198.846,Z 689.587,A -85,B 0,C 180,E1 8956.596,E2 8956.596} C_VEL
LIN {X 0,Y 194.793,Z 703.544,A -85,B 0,C 180,E1 8954.268,E2 8954.268} C_VEL
LIN {X 0,Y 190.047,Z 717.22,A -85,B 0,C 180,E1 8951.315,E2 8951.315} C_VEL
LIN {X 0,Y 185.29,Z 729.33,A -85,B 0,C 180,E1 8947.959,E2 8947.959} C_VEL
LIN {X 0,Y 180.544,Z 740.344,A -85,B 0,C 180,E1 8944.006,E2 8944.006} C_VEL
LIN {X 0,Y 176.281,Z 749.911,A -85,B 0,C 180,E1 8939.564,E2 8939.564} C_VEL
LIN {X 0,Y 172.725,Z 757.893,A -85,B 0,C 180,E1 8934.628,E2 8934.628} C_VEL
LIN {X 0,Y 170.117,Z 764.366,A -85,B 0,C 180,E1 8929.212,E2 8929.212} C_VEL
LIN {X 0,Y 168.648,Z 768.824,A -85,B 0,C 180,E1 8923.714,E2 8923.714} C_VEL
LIN {X 0,Y 168.195,Z 771.522,A -85,B 0,C 180,E1 8918.199,E2 8918.199} C_VEL
LIN {X 0,Y 168.288,Z 772.462,A -85,B 0,C 180,E1 8913.061,E2 8913.061} C_VEL
LIN {X 0,Y 168.371,Z 771.977,A -85,B 0,C 180,E1 8908.635,E2 8908.635} C_VEL
LIN {X 0,Y 168.323,Z 770.081,A -85,B 0,C 180,E1 8903.858,E2 8903.858} C_VEL
LIN {X 0,Y 168.303,Z 769.82,A -85,B 0,C 180,E1 8902.486,E2 8902.486} C_VEL
LIN {X 0,Y 168.793,Z 770.229,A -85,B 0,C 180,E1 8895.24,E2 8895.24} C_VEL
LIN {X 0,Y 171.509,Z 768.983,A -85,B 0,C 180,E1 8887.729,E2 8887.729} C_VEL
LIN {X 0,Y 177.821,Z 765.679,A -85,B 0,C 180,E1 8879.595,E2 8879.595} C_VEL
LIN {X 0,Y 188.556,Z 760.188,A -85,B 0,C 180,E1 8871.65,E2 8871.65} C_VEL
LIN {X 0,Y 203.653,Z 752.741,A -85,B 0,C 180,E1 8864.607,E2 8864.607} C_VEL
LIN {X 0,Y 211.316,Z 749.021,A -85,B 0,C 180,E1 8861.929,E2 8861.929} C_VEL
LIN {X 0,Y 196.422,Z 753.766,A -85,B 0,C 180,E1 8856.19,E2 8856.19} C_VEL
LIN {X 0,Y 184.626,Z 756.871,A -85,B 0,C 180,E1 8849.525,E2 8849.525} C_VEL
LIN {X 0,Y 176.34,Z 758.119,A -85,B 0,C 180,E1 8842.326,E2 8842.326} C_VEL
LIN {X 0,Y 171.293,Z 757.505,A -85,B 0,C 180,E1 8834.881,E2 8834.881} C_VEL
LIN {X 0,Y 168.972,Z 755.218,A -85,B 0,C 180,E1 8827.821,E2 8827.821} C_VEL
LIN {X 0,Y 168.29,Z 751.818,A -85,B 0,C 180,E1 8821.701,E2 8821.701} C_VEL
LIN {X 0,Y 168.197,Z 747.451,A -85,B 0,C 180,E1 8816.25,E2 8816.25} C_VEL
LIN {X 0,Y 168.584,Z 741.268,A -85,B 0,C 180,E1 8810.44,E2 8810.44} C_VEL
LIN {X 0,Y 169.788,Z 733.311,A -85,B 0,C 180,E1 8804.632,E2 8804.632} C_VEL
LIN {X 0,Y 172.098,Z 723.356,A -85,B 0,C 180,E1 8798.886,E2 8798.886} C_VEL
LIN {X 0,Y 175.56,Z 711.417,A -85,B 0,C 180,E1 8793.406,E2 8793.406} C_VEL
LIN {X 0,Y 179.882,Z 698.076,A -85,B 0,C 180,E1 8788.499,E2 8788.499} C_VEL
LIN {X 0,Y 184.919,Z 683.09,A -85,B 0,C 180,E1 8784.078,E2 8784.078} C_VEL
LIN {X 0,Y 190.431,Z 666.536,A -85,B 0,C 180,E1 8780.165,E2 8780.165} C_VEL
LIN {X 0,Y 196.007,Z 648.874,A -85,B 0,C 180,E1 8776.845,E2 8776.845} C_VEL
LIN {X 0,Y 201.591,Z 629.624,A -85,B 0,C 180,E1 8773.981,E2 8773.981} C_VEL
LIN {X 0,Y 207.04,Z 608.516,A -85,B 0,C 180,E1 8771.534,E2 8771.534} C_VEL
LIN {X 0,Y 211.706,Z 587.34,A -85,B 0,C 180,E1 8769.66,E2 8769.66} C_VEL
LIN {X 0,Y 215.64,Z 565.396,A -85,B 0,C 180,E1 8768.246,E2 8768.246} C_VEL
LIN {X 0,Y 234.928,Z 427.617,A -85,B 0,C 180,E1 8762.143,E2 8762.143} C_VEL
LIN {X 0,Y 233.125,Z 424.133,A -85,B 0,C 180,E1 8761.481,E2 8761.481} C_VEL
LIN {X 0,Y 230.769,Z 425.807,A -85,B 0,C 180,E1 8761.064,E2 8761.064} C_VEL
LIN {X 0,Y 225.246,Z 433.176,A -85,B 0,C 180,E1 8760.33,E2 8760.33} C_VEL
LIN {X 0,Y 221.567,Z 436.319,A -85,B 0,C 180,E1 8759.69,E2 8759.69} C_VEL
LIN {X 0,Y 219.541,Z 437.961,A -85,B 0,C 180,E1 8759.167,E2 8759.167} C_VEL
LIN {X 0,Y 218.156,Z 442.528,A -85,B 0,C 180,E1 8758.47,E2 8758.47} C_VEL
LIN {X 0,Y 209.499,Z 487.735,A -85,B 0,C 180,E1 8752.699,E2 8752.699} C_VEL
LIN {X 0,Y 210.665,Z 518.818,A -85,B 0,C 180,E1 8750.919,E2 8750.919} C_VEL
LIN {X 0,Y 202.963,Z 633.554,A -85,B 0,C 180,E1 8747.195,E2 8747.195} C_VEL
LIN {X 0,Y 200.899,Z 650.257,A -85,B 0,C 180,E1 8746.144,E2 8746.144} C_VEL
LIN {X 0,Y 198.235,Z 665.159,A -85,B 0,C 180,E1 8744.76,E2 8744.76} C_VEL
LIN {X 0,Y 194.818,Z 679.656,A -85,B 0,C 180,E1 8742.903,E2 8742.903} C_VEL
LIN {X 0,Y 190.653,Z 694.187,A -85,B 0,C 180,E1 8740.427,E2 8740.427} C_VEL
LIN {X 0,Y 186.361,Z 706.922,A -85,B 0,C 180,E1 8737.556,E2 8737.556} C_VEL
LIN {X 0,Y 181.968,Z 718.732,A -85,B 0,C 180,E1 8734.1,E2 8734.1} C_VEL
LIN {X 0,Y 177.982,Z 728.651,A -85,B 0,C 180,E1 8730.309,E2 8730.309} C_VEL
LIN {X 0,Y 174.23,Z 737.787,A -85,B 0,C 180,E1 8725.725,E2 8725.725} C_VEL
LIN {X 0,Y 171.426,Z 744.822,A -85,B 0,C 180,E1 8720.943,E2 8720.943} C_VEL
LIN {X 0,Y 169.483,Z 750.379,A -85,B 0,C 180,E1 8715.658,E2 8715.658} C_VEL
LIN {X 0,Y 168.571,Z 753.881,A -85,B 0,C 180,E1 8710.581,E2 8710.581} C_VEL
LIN {X 0,Y 168.319,Z 755.89,A -85,B 0,C 180,E1 8705.059,E2 8705.059} C_VEL
LIN {X 0,Y 168.642,Z 756.21,A -85,B 0,C 180,E1 8699.743,E2 8699.743} C_VEL
LIN {X 0,Y 169.762,Z 754.819,A -85,B 0,C 180,E1 8694.337,E2 8694.337} C_VEL
LIN {X 0,Y 172.008,Z 751.682,A -85,B 0,C 180,E1 8688.945,E2 8688.945} C_VEL
LIN {X 0,Y 175.241,Z 747.035,A -85,B 0,C 180,E1 8684.041,E2 8684.041} C_VEL
LIN {X 0,Y 179.593,Z 740.487,A -85,B 0,C 180,E1 8679.304,E2 8679.304} C_VEL
LIN {X 0,Y 184.754,Z 732.288,A -85,B 0,C 180,E1 8675.007,E2 8675.007} C_VEL
LIN {X 0,Y 190.458,Z 722.323,A -85,B 0,C 180,E1 8671.169,E2 8671.169} C_VEL
LIN {X 0,Y 196.127,Z 711.358,A -85,B 0,C 180,E1 8667.972,E2 8667.972} C_VEL
LIN {X 0,Y 201.673,Z 698.951,A -85,B 0,C 180,E1 8665.239,E2 8665.239} C_VEL
LIN {X 0,Y 206.822,Z 685.498,A -85,B 0,C 180,E1 8662.979,E2 8662.979} C_VEL
LIN {X 0,Y 211.423,Z 670.576,A -85,B 0,C 180,E1 8661.118,E2 8661.118} C_VEL
LIN {X 0,Y 214.892,Z 656.116,A -85,B 0,C 180,E1 8659.783,E2 8659.783} C_VEL
LIN {X 0,Y 217.57,Z 640.183,A -85,B 0,C 180,E1 8658.763,E2 8658.763} C_VEL
LIN {X 0,Y 219.391,Z 621.387,A -85,B 0,C 180,E1 8658.038,E2 8658.038} C_VEL
LIN {X 0,Y 227.565,Z 519.665,A -85,B 0,C 180,E1 8655.001,E2 8655.001} C_VEL
LIN {X 0,Y 226.964,Z 491.665,A -85,B 0,C 180,E1 8652.985,E2 8652.985} C_VEL
LIN {X 0,Y 227.705,Z 486.476,A -85,B 0,C 180,E1 8652.426,E2 8652.426} C_VEL
LIN {X 0,Y 238.01,Z 442.856,A -85,B 0,C 180,E1 8647.12,E2 8647.12} C_VEL
LIN {X 0,Y 238.558,Z 440.651,A -85,B 0,C 180,E1 8646.854,E2 8646.854} C_VEL
LIN {X 0,Y 239.044,Z 437.188,A -85,B 0,C 180,E1 8646.225,E2 8646.225} C_VEL
LIN {X 0,Y 238.564,Z 433.691,A -85,B 0,C 180,E1 8645.077,E2 8645.077} C_VEL
LIN {X 0,Y 236.422,Z 427.479,A -85,B 0,C 180,E1 8642.04,E2 8642.04} C_VEL
LIN {X 0,Y 235.366,Z 419.825,A -85,B 0,C 180,E1 8638.54,E2 8638.54} C_VEL
LIN {X 0,Y 234.261,Z 414.19,A -85,B 0,C 180,E1 8635.104,E2 8635.104} C_VEL
LIN {X 0,Y 233.64,Z 409.636,A -85,B 0,C 180,E1 8631.302,E2 8631.302} C_VEL
LIN {X 0,Y 233.642,Z 406.373,A -85,B 0,C 180,E1 8626.64,E2 8626.64} C_VEL
LIN {X 0,Y 233.888,Z 406.188,A -85,B 0,C 180,E1 8622.589,E2 8622.589} C_VEL
LIN {X 0,Y 233.923,Z 406.605,A -85,B 0,C 180,E1 8622.077,E2 8622.077} C_VEL
LIN {X 0,Y 231.401,Z 422.323,A -85,B 0,C 180,E1 8616.344,E2 8616.344} C_VEL
LIN {X 0,Y 231.464,Z 426.766,A -85,B 0,C 180,E1 8614.836,E2 8614.836} C_VEL
LIN {X 0,Y 234.206,Z 432.58,A -85,B 0,C 180,E1 8613.766,E2 8613.766} C_VEL
LIN {X 0,Y 214.117,Z 574.365,A -85,B 0,C 180,E1 8607.702,E2 8607.702} C_VEL
LIN {X 0,Y 209.776,Z 596.826,A -85,B 0,C 180,E1 8606.27,E2 8606.27} C_VEL
LIN {X 0,Y 204.359,Z 619.531,A -85,B 0,C 180,E1 8604.303,E2 8604.303} C_VEL
LIN {X 0,Y 203.513,Z 624.212,A -85,B 0,C 180,E1 8603.995,E2 8603.995} C_VEL
LIN {X 0,Y 201.91,Z 648.108,A -85,B 0,C 180,E1 8602.761,E2 8602.761} C_VEL
LIN {X 0,Y 200,Z 662.648,A -85,B 0,C 180,E1 8601.647,E2 8601.647} C_VEL
LIN {X 0,Y 197.204,Z 676.915,A -85,B 0,C 180,E1 8600.18,E2 8600.18} C_VEL
LIN {X 0,Y 193.529,Z 691.091,A -85,B 0,C 180,E1 8598.287,E2 8598.287} C_VEL
LIN {X 0,Y 188.844,Z 705.51,A -85,B 0,C 180,E1 8595.76,E2 8595.76} C_VEL
LIN {X 0,Y 183.859,Z 718.529,A -85,B 0,C 180,E1 8592.82,E2 8592.82} C_VEL
LIN {X 0,Y 178.555,Z 730.688,A -85,B 0,C 180,E1 8589.25,E2 8589.25} C_VEL
LIN {X 0,Y 173.494,Z 741.383,A -85,B 0,C 180,E1 8585.186,E2 8585.186} C_VEL
LIN {X 0,Y 168.92,Z 750.58,A -85,B 0,C 180,E1 8580.596,E2 8580.596} C_VEL
LIN {X 0,Y 164.889,Z 758.8,A -85,B 0,C 180,E1 8575.112,E2 8575.112} C_VEL
LIN {X 0,Y 162.145,Z 764.84,A -85,B 0,C 180,E1 8569.446,E2 8569.446} C_VEL
LIN {X 0,Y 160.629,Z 769.021,A -85,B 0,C 180,E1 8563.678,E2 8563.678} C_VEL
LIN {X 0,Y 160.192,Z 771.404,A -85,B 0,C 180,E1 8557.889,E2 8557.889} C_VEL
LIN {X 0,Y 160.319,Z 772.033,A -85,B 0,C 180,E1 8552.498,E2 8552.498} C_VEL
LIN {X 0,Y 160.369,Z 771.303,A -85,B 0,C 180,E1 8547.852,E2 8547.852} C_VEL
LIN {X 0,Y 160.352,Z 768.92,A -85,B 0,C 180,E1 8542.112,E2 8542.112} C_VEL
LIN {X 0,Y 160.947,Z 769.601,A -85,B 0,C 180,E1 8534.503,E2 8534.503} C_VEL
LIN {X 0,Y 164.172,Z 768.537,A -85,B 0,C 180,E1 8526.295,E2 8526.295} C_VEL
LIN {X 0,Y 171.188,Z 765.587,A -85,B 0,C 180,E1 8517.874,E2 8517.874} C_VEL
LIN {X 0,Y 183.295,Z 760.405,A -85,B 0,C 180,E1 8509.52,E2 8509.52} C_VEL
LIN {X 0,Y 199.447,Z 753.565,A -85,B 0,C 180,E1 8502.525,E2 8502.525} C_VEL
LIN {X 0,Y 201.156,Z 752.825,A -85,B 0,C 180,E1 8501.858,E2 8501.858} C_VEL
LIN {X 0,Y 185.881,Z 756.616,A -85,B 0,C 180,E1 8495.515,E2 8495.515} C_VEL
LIN {X 0,Y 174.097,Z 758.634,A -85,B 0,C 180,E1 8488.094,E2 8488.094} C_VEL
LIN {X 0,Y 166.488,Z 758.702,A -85,B 0,C 180,E1 8480.384,E2 8480.384} C_VEL
LIN {X 0,Y 162.328,Z 757.034,A -85,B 0,C 180,E1 8472.81,E2 8472.81} C_VEL
LIN {X 0,Y 160.621,Z 753.914,A -85,B 0,C 180,E1 8465.715,E2 8465.715} C_VEL
LIN {X 0,Y 160.227,Z 749.933,A -85,B 0,C 180,E1 8459.641,E2 8459.641} C_VEL
LIN {X 0,Y 160.288,Z 744.773,A -85,B 0,C 180,E1 8453.911,E2 8453.911} C_VEL
LIN {X 0,Y 161.003,Z 737.672,A -85,B 0,C 180,E1 8447.809,E2 8447.809} C_VEL
LIN {X 0,Y 162.736,Z 728.688,A -85,B 0,C 180,E1 8441.738,E2 8441.738} C_VEL
LIN {X 0,Y 165.518,Z 718.279,A -85,B 0,C 180,E1 8436.124,E2 8436.124} C_VEL
LIN {X 0,Y 169.491,Z 705.708,A -85,B 0,C 180,E1 8430.682,E2 8430.682} C_VEL
LIN {X 0,Y 174.318,Z 691.587,A -85,B 0,C 180,E1 8425.796,E2 8425.796} C_VEL
LIN {X 0,Y 179.96,Z 675.353,A -85,B 0,C 180,E1 8421.312,E2 8421.312} C_VEL
LIN {X 0,Y 185.561,Z 658.707,A -85,B 0,C 180,E1 8417.658,E2 8417.658} C_VEL
LIN {X 0,Y 191.569,Z 639.598,A -85,B 0,C 180,E1 8414.351,E2 8414.351} C_VEL
LIN {X 0,Y 197.398,Z 619.056,A -85,B 0,C 180,E1 8411.574,E2 8411.574} C_VEL
LIN {X 0,Y 202.545,Z 598.322,A -85,B 0,C 180,E1 8409.414,E2 8409.414} C_VEL
LIN {X 0,Y 207.089,Z 576.326,A -85,B 0,C 180,E1 8407.699,E2 8407.699} C_VEL
LIN {X 0,Y 211.001,Z 551.851,A -85,B 0,C 180,E1 8406.354,E2 8406.354} C_VEL
LIN {X 0,Y 227.233,Z 440.079,A -85,B 0,C 180,E1 8401.325,E2 8401.325} C_VEL
LIN {X 0,Y 222.58,Z 443.633,A -85,B 0,C 180,E1 8400.508,E2 8400.508} C_VEL
LIN {X 0,Y 221.414,Z 444.853,A -85,B 0,C 180,E1 8400.33,E2 8400.33} C_VEL
LIN {X 0,Y 216.084,Z 451.918,A -85,B 0,C 180,E1 8399.611,E2 8399.611} C_VEL
LIN {X 0,Y 212.316,Z 455.133,A -85,B 0,C 180,E1 8398.942,E2 8398.942} C_VEL
LIN {X 0,Y 210.266,Z 456.816,A -85,B 0,C 180,E1 8398.396,E2 8398.396} C_VEL
LIN {X 0,Y 208.844,Z 461.49,A -85,B 0,C 180,E1 8397.674,E2 8397.674} C_VEL
LIN {X 0,Y 203.614,Z 488.758,A -85,B 0,C 180,E1 8394.178,E2 8394.178} C_VEL
LIN {X 0,Y 204.632,Z 519.551,A -85,B 0,C 180,E1 8392.363,E2 8392.363} C_VEL
LIN {X 0,Y 196.623,Z 633.934,A -85,B 0,C 180,E1 8388.591,E2 8388.591} C_VEL
LIN {X 0,Y 194.482,Z 650.561,A -85,B 0,C 180,E1 8387.525,E2 8387.525} C_VEL
LIN {X 0,Y 191.599,Z 665.988,A -85,B 0,C 180,E1 8386.059,E2 8386.059} C_VEL
LIN {X 0,Y 187.788,Z 681.269,A -85,B 0,C 180,E1 8384.023,E2 8384.023} C_VEL
LIN {X 0,Y 183.461,Z 695.537,A -85,B 0,C 180,E1 8381.477,E2 8381.477} C_VEL
LIN {X 0,Y 178.786,Z 708.651,A -85,B 0,C 180,E1 8378.364,E2 8378.364} C_VEL
LIN {X 0,Y 174.426,Z 719.757,A -85,B 0,C 180,E1 8374.936,E2 8374.936} C_VEL
LIN {X 0,Y 169.976,Z 730.229,A -85,B 0,C 180,E1 8370.678,E2 8370.678} C_VEL
LIN {X 0,Y 166.35,Z 738.634,A -85,B 0,C 180,E1 8366.184,E2 8366.184} C_VEL
LIN {X 0,Y 163.459,Z 745.511,A -85,B 0,C 180,E1 8361.208,E2 8361.208} C_VEL
LIN {X 0,Y 161.462,Z 750.998,A -85,B 0,C 180,E1 8355.663,E2 8355.663} C_VEL
LIN {X 0,Y 160.513,Z 754.566,A -85,B 0,C 180,E1 8349.969,E2 8349.969} C_VEL
LIN {X 0,Y 160.333,Z 756.348,A -85,B 0,C 180,E1 8344.518,E2 8344.518} C_VEL
LIN {X 0,Y 160.754,Z 756.579,A -85,B 0,C 180,E1 8338.924,E2 8338.924} C_VEL
LIN {X 0,Y 162.224,Z 754.933,A -85,B 0,C 180,E1 8332.847,E2 8332.847} C_VEL
LIN {X 0,Y 164.898,Z 751.567,A -85,B 0,C 180,E1 8327.198,E2 8327.198} C_VEL
LIN {X 0,Y 168.893,Z 746.228,A -85,B 0,C 180,E1 8321.768,E2 8321.768} C_VEL
LIN {X 0,Y 173.835,Z 739.315,A -85,B 0,C 180,E1 8316.925,E2 8316.925} C_VEL
LIN {X 0,Y 179.748,Z 730.328,A -85,B 0,C 180,E1 8312.444,E2 8312.444} C_VEL
LIN {X 0,Y 185.805,Z 720.142,A -85,B 0,C 180,E1 8308.709,E2 8308.709} C_VEL
LIN {X 0,Y 192.09,Z 708.2,A -85,B 0,C 180,E1 8305.44,E2 8305.44} C_VEL
LIN {X 0,Y 197.59,Z 696.12,A -85,B 0,C 180,E1 8302.933,E2 8302.933} C_VEL
LIN {X 0,Y 203.058,Z 681.742,A -85,B 0,C 180,E1 8300.692,E2 8300.692} C_VEL
LIN {X 0,Y 207.513,Z 667.094,A -85,B 0,C 180,E1 8298.999,E2 8298.999} C_VEL
LIN {X 0,Y 211.229,Z 650.564,A -85,B 0,C 180,E1 8297.636,E2 8297.636} C_VEL
LIN {X 0,Y 213.589,Z 634.573,A -85,B 0,C 180,E1 8296.766,E2 8296.766} C_VEL
LIN {X 0,Y 223.224,Z 520.734,A -85,B 0,C 180,E1 8293.305,E2 8293.305} C_VEL
LIN {X 0,Y 222.906,Z 493.056,A -85,B 0,C 180,E1 8291.253,E2 8291.253} C_VEL
LIN {X 0,Y 223.234,Z 488.794,A -85,B 0,C 180,E1 8290.844,E2 8290.844} C_VEL
LIN {X 0,Y 233.54,Z 447.232,A -85,B 0,C 180,E1 8285.775,E2 8285.775} C_VEL
LIN {X 0,Y 237.089,Z 432.81,A -85,B 0,C 180,E1 8283.991,E2 8283.991} C_VEL
LIN {X 0,Y 236.422,Z 427.479,A -85,B 0,C 180,E1 8282.04,E2 8282.04} C_VEL
LIN {X 0,Y 235.623,Z 424.837,A -85,B 0,C 180,E1 8280.575,E2 8280.575} C_VEL
LIN {X 0,Y 233.667,Z 422.928,A -85,B 0,C 180,E1 8278.21,E2 8278.21} C_VEL
LIN {X 0,Y 231.182,Z 421.007,A -85,B 0,C 180,E1 8274.645,E2 8274.645} C_VEL
LIN {X 0,Y 230.926,Z 419.801,A -85,B 0,C 180,E1 8273.563,E2 8273.563} C_VEL
LIN {X 0,Y 230.46,Z 416.606,A -85,B 0,C 180,E1 8270.512,E2 8270.512} C_VEL
LIN {X 0,Y 230.78,Z 413.806,A -85,B 0,C 180,E1 8266.215,E2 8266.215} C_VEL
LIN {X 0,Y 231.018,Z 413.815,A -85,B 0,C 180,E1 8262.755,E2 8262.755} C_VEL
LIN {X 0,Y 228.173,Z 430.939,A -85,B 0,C 180,E1 8256.5,E2 8256.5} C_VEL
LIN {X 0,Y 228.012,Z 435.468,A -85,B 0,C 180,E1 8255.029,E2 8255.029} C_VEL
LIN {X 0,Y 207.408,Z 574.805,A -85,B 0,C 180,E1 8248.895,E2 8248.895} C_VEL
LIN {X 0,Y 202.897,Z 597.264,A -85,B 0,C 180,E1 8247.417,E2 8247.417} C_VEL
LIN {X 0,Y 201.248,Z 605.535,A -85,B 0,C 180,E1 8246.864,E2 8246.864} C_VEL
LIN {X 0,Y 200.055,Z 621.802,A -85,B 0,C 180,E1 8246.129,E2 8246.129} C_VEL
LIN {X 0,Y 199.017,Z 637.587,A -85,B 0,C 180,E1 8245.36,E2 8245.36} C_VEL
LIN {X 0,Y 197.793,Z 650.252,A -85,B 0,C 180,E1 8244.64,E2 8244.64} C_VEL
LIN {X 0,Y 195.668,Z 663.933,A -85,B 0,C 180,E1 8243.56,E2 8243.56} C_VEL
LIN {X 0,Y 192.609,Z 677.955,A -85,B 0,C 180,E1 8242.091,E2 8242.091} C_VEL
LIN {X 0,Y 188.65,Z 691.693,A -85,B 0,C 180,E1 8240.214,E2 8240.214} C_VEL
LIN {X 0,Y 183.485,Z 706.278,A -85,B 0,C 180,E1 8237.602,E2 8237.602} C_VEL
LIN {X 0,Y 178.044,Z 719.249,A -85,B 0,C 180,E1 8234.58,E2 8234.58} C_VEL
LIN {X 0,Y 172.357,Z 731.173,A -85,B 0,C 180,E1 8230.954,E2 8230.954} C_VEL
LIN {X 0,Y 166.901,Z 741.673,A -85,B 0,C 180,E1 8226.798,E2 8226.798} C_VEL
LIN {X 0,Y 161.621,Z 751.27,A -85,B 0,C 180,E1 8221.72,E2 8221.72} C_VEL
LIN {X 0,Y 157.511,Z 758.77,A -85,B 0,C 180,E1 8216.377,E2 8216.377} C_VEL
LIN {X 0,Y 154.463,Z 764.695,A -85,B 0,C 180,E1 8210.455,E2 8210.455} C_VEL
LIN {X 0,Y 152.725,Z 768.827,A -85,B 0,C 180,E1 8204.326,E2 8204.326} C_VEL
LIN {X 0,Y 152.201,Z 771.06,A -85,B 0,C 180,E1 8198.306,E2 8198.306} C_VEL
LIN {X 0,Y 152.323,Z 771.623,A -85,B 0,C 180,E1 8192.629,E2 8192.629} C_VEL
LIN {X 0,Y 152.378,Z 770.824,A -85,B 0,C 180,E1 8187.74,E2 8187.74} C_VEL
LIN {X 0,Y 152.369,Z 768.382,A -85,B 0,C 180,E1 8182.075,E2 8182.075} C_VEL
LIN {X 0,Y 152.403,Z 768.051,A -85,B 0,C 180,E1 8180.937,E2 8180.937} C_VEL
LIN {X 0,Y 153.327,Z 768.816,A -85,B 0,C 180,E1 8172.931,E2 8172.931} C_VEL
LIN {X 0,Y 157.422,Z 767.916,A -85,B 0,C 180,E1 8164.004,E2 8164.004} C_VEL
LIN {X 0,Y 166.294,Z 764.952,A -85,B 0,C 180,E1 8154.741,E2 8154.741} C_VEL
LIN {X 0,Y 179.981,Z 760.058,A -85,B 0,C 180,E1 8146.456,E2 8146.456} C_VEL
LIN {X 0,Y 190.979,Z 756.033,A -85,B 0,C 180,E1 8141.795,E2 8141.795} C_VEL
LIN {X 0,Y 175.669,Z 758.775,A -85,B 0,C 180,E1 8134.949,E2 8134.949} C_VEL
LIN {X 0,Y 164.759,Z 759.68,A -85,B 0,C 180,E1 8127.464,E2 8127.464} C_VEL
LIN {X 0,Y 157.483,Z 758.803,A -85,B 0,C 180,E1 8119.276,E2 8119.276} C_VEL
LIN {X 0,Y 153.749,Z 756.259,A -85,B 0,C 180,E1 8111.249,E2 8111.249} C_VEL
LIN {X 0,Y 152.428,Z 752.31,A -85,B 0,C 180,E1 8103.76,E2 8103.76} C_VEL
LIN {X 0,Y 152.211,Z 747.873,A -85,B 0,C 180,E1 8097.74,E2 8097.74} C_VEL
LIN {X 0,Y 152.462,Z 741.959,A -85,B 0,C 180,E1 8091.703,E2 8091.703} C_VEL
LIN {X 0,Y 153.556,Z 733.994,A -85,B 0,C 180,E1 8085.288,E2 8085.288} C_VEL
LIN {X 0,Y 155.863,Z 724.042,A -85,B 0,C 180,E1 8078.945,E2 8078.945} C_VEL
LIN {X 0,Y 159.422,Z 712.205,A -85,B 0,C 180,E1 8072.955,E2 8072.955} C_VEL
LIN {X 0,Y 164.001,Z 698.806,A -85,B 0,C 180,E1 8067.552,E2 8067.552} C_VEL
LIN {X 0,Y 169.34,Z 683.884,A -85,B 0,C 180,E1 8062.755,E2 8062.755} C_VEL
LIN {X 0,Y 175.192,Z 667.429,A -85,B 0,C 180,E1 8058.543,E2 8058.543} C_VEL
LIN {X 0,Y 181.263,Z 649.43,A -85,B 0,C 180,E1 8054.919,E2 8054.919} C_VEL
LIN {X 0,Y 187.216,Z 630.282,A -85,B 0,C 180,E1 8051.884,E2 8051.884} C_VEL
LIN {X 0,Y 193.011,Z 609.33,A -85,B 0,C 180,E1 8049.308,E2 8049.308} C_VEL
LIN {X 0,Y 198.029,Z 588.042,A -85,B 0,C 180,E1 8047.321,E2 8047.321} C_VEL
LIN {X 0,Y 202.331,Z 565.771,A -85,B 0,C 180,E1 8045.805,E2 8045.805} C_VEL
LIN {X 0,Y 218.439,Z 458.466,A -85,B 0,C 180,E1 8040.707,E2 8040.707} C_VEL
LIN {X 0,Y 213.978,Z 462.059,A -85,B 0,C 180,E1 8039.924,E2 8039.924} C_VEL
LIN {X 0,Y 212.508,Z 463.195,A -85,B 0,C 180,E1 8039.661,E2 8039.661} C_VEL
LIN {X 0,Y 207.004,Z 470.589,A -85,B 0,C 180,E1 8038.925,E2 8038.925} C_VEL
LIN {X 0,Y 203.137,Z 473.924,A -85,B 0,C 180,E1 8038.228,E2 8038.228} C_VEL
LIN {X 0,Y 201.131,Z 475.381,A -85,B 0,C 180,E1 8037.701,E2 8037.701} C_VEL
LIN {X 0,Y 199.828,Z 478.864,A -85,B 0,C 180,E1 8037.089,E2 8037.089} C_VEL
LIN {X 0,Y 197.861,Z 489.188,A -85,B 0,C 180,E1 8035.782,E2 8035.782} C_VEL
LIN {X 0,Y 198.705,Z 520.426,A -85,B 0,C 180,E1 8033.884,E2 8033.884} C_VEL
LIN {X 0,Y 190.39,Z 634.283,A -85,B 0,C 180,E1 8030.073,E2 8030.073} C_VEL
LIN {X 0,Y 188.148,Z 650.98,A -85,B 0,C 180,E1 8028.985,E2 8028.985} C_VEL
LIN {X 0,Y 185.065,Z 666.733,A -85,B 0,C 180,E1 8027.452,E2 8027.452} C_VEL
LIN {X 0,Y 181.093,Z 681.937,A -85,B 0,C 180,E1 8025.372,E2 8025.372} C_VEL
LIN {X 0,Y 176.819,Z 695.455,A -85,B 0,C 180,E1 8022.91,E2 8022.91} C_VEL
LIN {X 0,Y 171.909,Z 708.656,A -85,B 0,C 180,E1 8019.714,E2 8019.714} C_VEL
LIN {X 0,Y 167.314,Z 719.842,A -85,B 0,C 180,E1 8016.179,E2 8016.179} C_VEL
LIN {X 0,Y 162.608,Z 730.379,A -85,B 0,C 180,E1 8011.766,E2 8011.766} C_VEL
LIN {X 0,Y 158.779,Z 738.788,A -85,B 0,C 180,E1 8007.116,E2 8007.116} C_VEL
LIN {X 0,Y 155.602,Z 745.937,A -85,B 0,C 180,E1 8001.726,E2 8001.726} C_VEL
LIN {X 0,Y 153.529,Z 751.319,A -85,B 0,C 180,E1 7996.023,E2 7996.023} C_VEL
LIN {X 0,Y 152.525,Z 754.902,A -85,B 0,C 180,E1 7990.074,E2 7990.074} C_VEL
LIN {X 0,Y 152.349,Z 756.776,A -85,B 0,C 180,E1 7984.046,E2 7984.046} C_VEL
LIN {X 0,Y 152.859,Z 756.971,A -85,B 0,C 180,E1 7978.251,E2 7978.251} C_VEL
LIN {X 0,Y 154.466,Z 755.389,A -85,B 0,C 180,E1 7972.058,E2 7972.058} C_VEL
LIN {X 0,Y 157.379,Z 752.102,A -85,B 0,C 180,E1 7966.178,E2 7966.178} C_VEL
LIN {X 0,Y 161.744,Z 746.766,A -85,B 0,C 180,E1 7960.474,E2 7960.474} C_VEL
LIN {X 0,Y 167.015,Z 739.953,A -85,B 0,C 180,E1 7955.501,E2 7955.501} C_VEL
LIN {X 0,Y 173.311,Z 731.031,A -85,B 0,C 180,E1 7950.896,E2 7950.896} C_VEL
LIN {X 0,Y 179.697,Z 721.022,A -85,B 0,C 180,E1 7947.103,E2 7947.103} C_VEL
LIN {X 0,Y 185.971,Z 709.823,A -85,B 0,C 180,E1 7943.947,E2 7943.947} C_VEL
LIN {X 0,Y 192.047,Z 697.314,A -85,B 0,C 180,E1 7941.273,E2 7941.273} C_VEL
LIN {X 0,Y 197.355,Z 684.211,A -85,B 0,C 180,E1 7939.171,E2 7939.171} C_VEL
LIN {X 0,Y 202.206,Z 669.444,A -85,B 0,C 180,E1 7937.394,E2 7937.394} C_VEL
LIN {X 0,Y 205.999,Z 654.08,A -85,B 0,C 180,E1 7936.061,E2 7936.061} C_VEL
LIN {X 0,Y 208.829,Z 637.258,A -85,B 0,C 180,E1 7935.072,E2 7935.072} C_VEL
LIN {X 0,Y 213.017,Z 590.957,A -85,B 0,C 180,E1 7933.594,E2 7933.594} C_VEL
LIN {X 0,Y 219.172,Z 521.821,A -85,B 0,C 180,E1 7931.53,E2 7931.53} C_VEL
LIN {X 0,Y 219.13,Z 494.343,A -85,B 0,C 180,E1 7929.439,E2 7929.439} C_VEL
LIN {X 0,Y 219.29,Z 489.996,A -85,B 0,C 180,E1 7929.051,E2 7929.051} C_VEL
LIN {X 0,Y 230.062,Z 448.378,A -85,B 0,C 180,E1 7923.988,E2 7923.988} C_VEL
LIN {X 0,Y 232.935,Z 437.369,A -85,B 0,C 180,E1 7922.646,E2 7922.646} C_VEL
LIN {X 0,Y 232.182,Z 429.752,A -85,B 0,C 180,E1 7919.507,E2 7919.507} C_VEL
LIN {X 0,Y 231.38,Z 424.088,A -85,B 0,C 180,E1 7916.521,E2 7916.521} C_VEL
LIN {X 0,Y 230.926,Z 419.801,A -85,B 0,C 180,E1 7913.563,E2 7913.563} C_VEL
LIN {X 0,Y 230.574,Z 418.534,A -85,B 0,C 180,E1 7911.953,E2 7911.953} C_VEL
LIN {X 0,Y 229.588,Z 418.914,A -85,B 0,C 180,E1 7909.61,E2 7909.61} C_VEL
LIN {X 0,Y 228.041,Z 421.125,A -85,B 0,C 180,E1 7905.376,E2 7905.376} C_VEL
LIN {X 0,Y 227.979,Z 421.154,A -85,B 0,C 180,E1 7904.659,E2 7904.659} C_VEL
LIN {X 0,Y 228.094,Z 421.22,A -85,B 0,C 180,E1 7903.381,E2 7903.381} C_VEL
LIN {X 0,Y 225.005,Z 438.69,A -85,B 0,C 180,E1 7896.981,E2 7896.981} C_VEL
LIN {X 0,Y 224.901,Z 439.395,A -85,B 0,C 180,E1 7896.795,E2 7896.795} C_VEL
LIN {X 0,Y 217.624,Z 464.44,A -85,B 0,C 180,E1 7895.247,E2 7895.247} C_VEL
LIN {X 0,Y 200.394,Z 578.791,A -85,B 0,C 180,E1 7890.059,E2 7890.059} C_VEL
LIN {X 0,Y 198.399,Z 601.252,A -85,B 0,C 180,E1 7889.173,E2 7889.173} C_VEL
LIN {X 0,Y 196.659,Z 622.745,A -85,B 0,C 180,E1 7888.206,E2 7888.206} C_VEL
LIN {X 0,Y 194.44,Z 647.901,A -85,B 0,C 180,E1 7886.942,E2 7886.942} C_VEL
LIN {X 0,Y 191.865,Z 663.877,A -85,B 0,C 180,E1 7885.702,E2 7885.702} C_VEL
LIN {X 0,Y 188.236,Z 678.98,A -85,B 0,C 180,E1 7884.093,E2 7884.093} C_VEL
LIN {X 0,Y 183.539,Z 693.743,A -85,B 0,C 180,E1 7882.007,E2 7882.007} C_VEL
LIN {X 0,Y 178.346,Z 707.121,A -85,B 0,C 180,E1 7879.55,E2 7879.55} C_VEL
LIN {X 0,Y 172.064,Z 720.719,A -85,B 0,C 180,E1 7876.252,E2 7876.252} C_VEL
LIN {X 0,Y 165.86,Z 732.583,A -85,B 0,C 180,E1 7872.462,E2 7872.462} C_VEL
LIN {X 0,Y 159.63,Z 743.349,A -85,B 0,C 180,E1 7867.862,E2 7867.862} C_VEL
LIN {X 0,Y 154.392,Z 751.973,A -85,B 0,C 180,E1 7862.951,E2 7862.951} C_VEL
LIN {X 0,Y 149.964,Z 759.156,A -85,B 0,C 180,E1 7857.385,E2 7857.385} C_VEL
LIN {X 0,Y 146.667,Z 764.871,A -85,B 0,C 180,E1 7851.176,E2 7851.176} C_VEL
LIN {X 0,Y 144.791,Z 768.714,A -85,B 0,C 180,E1 7844.799,E2 7844.799} C_VEL
LIN {X 0,Y 144.205,Z 770.801,A -85,B 0,C 180,E1 7838.368,E2 7838.368} C_VEL
LIN {X 0,Y 144.327,Z 771.212,A -85,B 0,C 180,E1 7832.775,E2 7832.775} C_VEL
LIN {X 0,Y 144.394,Z 770.455,A -85,B 0,C 180,E1 7828.012,E2 7828.012} C_VEL
LIN {X 0,Y 144.368,Z 768.226,A -85,B 0,C 180,E1 7822.434,E2 7822.434} C_VEL
LIN {X 0,Y 144.49,Z 767.034,A -85,B 0,C 180,E1 7820.034,E2 7820.034} C_VEL
LIN {X 0,Y 145.948,Z 768.02,A -85,B 0,C 180,E1 7810.798,E2 7810.798} C_VEL
LIN {X 0,Y 151.239,Z 767.234,A -85,B 0,C 180,E1 7801.14,E2 7801.14} C_VEL
LIN {X 0,Y 161.503,Z 764.512,A -85,B 0,C 180,E1 7791.746,E2 7791.746} C_VEL
LIN {X 0,Y 176.639,Z 760.01,A -85,B 0,C 180,E1 7783.565,E2 7783.565} C_VEL
LIN {X 0,Y 180.856,Z 758.644,A -85,B 0,C 180,E1 7781.772,E2 7781.772} C_VEL
LIN {X 0,Y 166.303,Z 760.289,A -85,B 0,C 180,E1 7774.83,E2 7774.83} C_VEL
LIN {X 0,Y 155.426,Z 760.26,A -85,B 0,C 180,E1 7766.762,E2 7766.762} C_VEL
LIN {X 0,Y 148.532,Z 758.45,A -85,B 0,C 180,E1 7758.037,E2 7758.037} C_VEL
LIN {X 0,Y 145.264,Z 755.031,A -85,B 0,C 180,E1 7749.507,E2 7749.507} C_VEL
LIN {X 0,Y 144.339,Z 750.518,A -85,B 0,C 180,E1 7741.983,E2 7741.983} C_VEL
LIN {X 0,Y 144.254,Z 745.363,A -85,B 0,C 180,E1 7735.626,E2 7735.626} C_VEL
LIN {X 0,Y 144.765,Z 738.683,A -85,B 0,C 180,E1 7729.251,E2 7729.251} C_VEL
LIN {X 0,Y 146.359,Z 729.797,A -85,B 0,C 180,E1 7722.506,E2 7722.506} C_VEL
LIN {X 0,Y 149.333,Z 718.796,A -85,B 0,C 180,E1 7715.893,E2 7715.893} C_VEL
LIN {X 0,Y 153.499,Z 706.229,A -85,B 0,C 180,E1 7709.895,E2 7709.895} C_VEL
LIN {X 0,Y 158.616,Z 692.123,A -85,B 0,C 180,E1 7704.552,E2 7704.552} C_VEL
LIN {X 0,Y 164.624,Z 675.94,A -85,B 0,C 180,E1 7699.695,E2 7699.695} C_VEL
LIN {X 0,Y 170.871,Z 658.525,A -85,B 0,C 180,E1 7695.607,E2 7695.607} C_VEL
LIN {X 0,Y 177.259,Z 639.518,A -85,B 0,C 180,E1 7692.118,E2 7692.118} C_VEL
LIN {X 0,Y 183.384,Z 619.315,A -85,B 0,C 180,E1 7689.236,E2 7689.236} C_VEL
LIN {X 0,Y 188.924,Z 598.368,A -85,B 0,C 180,E1 7686.949,E2 7686.949} C_VEL
LIN {X 0,Y 193.811,Z 576.226,A -85,B 0,C 180,E1 7685.144,E2 7685.144} C_VEL
LIN {X 0,Y 198.126,Z 551.12,A -85,B 0,C 180,E1 7683.695,E2 7683.695} C_VEL
LIN {X 0,Y 209.631,Z 476.889,A -85,B 0,C 180,E1 7680.108,E2 7680.108} C_VEL
LIN {X 0,Y 205.044,Z 480.699,A -85,B 0,C 180,E1 7679.304,E2 7679.304} C_VEL
LIN {X 0,Y 203.21,Z 482.007,A -85,B 0,C 180,E1 7678.958,E2 7678.958} C_VEL
LIN {X 0,Y 197.545,Z 489.63,A -85,B 0,C 180,E1 7678.195,E2 7678.195} C_VEL
LIN {X 0,Y 193.811,Z 493.658,A -85,B 0,C 180,E1 7677.551,E2 7677.551} C_VEL
LIN {X 0,Y 192.684,Z 496.1,A -85,B 0,C 180,E1 7677.132,E2 7677.132} C_VEL
LIN {X 0,Y 192.749,Z 509.195,A -85,B 0,C 180,E1 7676.214,E2 7676.214} C_VEL
LIN {X 0,Y 192.907,Z 521.389,A -85,B 0,C 180,E1 7675.489,E2 7675.489} C_VEL
LIN {X 0,Y 184.25,Z 634.762,A -85,B 0,C 180,E1 7671.637,E2 7671.637} C_VEL
LIN {X 0,Y 181.903,Z 651.472,A -85,B 0,C 180,E1 7670.527,E2 7670.527} C_VEL
LIN {X 0,Y 178.643,Z 667.365,A -85,B 0,C 180,E1 7668.946,E2 7668.946} C_VEL
LIN {X 0,Y 174.391,Z 682.892,A -85,B 0,C 180,E1 7666.763,E2 7666.763} C_VEL
LIN {X 0,Y 169.782,Z 696.676,A -85,B 0,C 180,E1 7664.15,E2 7664.15} C_VEL
LIN {X 0,Y 164.438,Z 710.307,A -85,B 0,C 180,E1 7660.691,E2 7660.691} C_VEL
LIN {X 0,Y 159.461,Z 721.651,A -85,B 0,C 180,E1 7656.846,E2 7656.846} C_VEL
LIN {X 0,Y 154.615,Z 731.945,A -85,B 0,C 180,E1 7652.228,E2 7652.228} C_VEL
LIN {X 0,Y 150.686,Z 740.07,A -85,B 0,C 180,E1 7647.342,E2 7647.342} C_VEL
LIN {X 0,Y 147.355,Z 747.278,A -85,B 0,C 180,E1 7641.419,E2 7641.419} C_VEL
LIN {X 0,Y 145.412,Z 752.155,A -85,B 0,C 180,E1 7635.673,E2 7635.673} C_VEL
LIN {X 0,Y 144.455,Z 755.672,A -85,B 0,C 180,E1 7629.138,E2 7629.138} C_VEL
LIN {X 0,Y 144.383,Z 757.254,A -85,B 0,C 180,E1 7623.253,E2 7623.253} C_VEL
LIN {X 0,Y 145.069,Z 757.297,A -85,B 0,C 180,E1 7617.016,E2 7617.016} C_VEL
LIN {X 0,Y 147.107,Z 755.522,A -85,B 0,C 180,E1 7610.296,E2 7610.296} C_VEL
LIN {X 0,Y 150.512,Z 751.971,A -85,B 0,C 180,E1 7604.162,E2 7604.162} C_VEL
LIN {X 0,Y 155.429,Z 746.493,A -85,B 0,C 180,E1 7598.304,E2 7598.304} C_VEL
LIN {X 0,Y 161.284,Z 739.378,A -85,B 0,C 180,E1 7593.193,E2 7593.193} C_VEL
LIN {X 0,Y 168.033,Z 730.398,A -85,B 0,C 180,E1 7588.606,E2 7588.606} C_VEL
LIN {X 0,Y 174.741,Z 720.288,A -85,B 0,C 180,E1 7584.868,E2 7584.868} C_VEL
LIN {X 0,Y 181.709,Z 708.335,A -85,B 0,C 180,E1 7581.588,E2 7581.588} C_VEL
LIN {X 0,Y 188.141,Z 695.233,A -85,B 0,C 180,E1 7578.934,E2 7578.934} C_VEL
LIN {X 0,Y 193.986,Z 680.931,A -85,B 0,C 180,E1 7576.778,E2 7576.778} C_VEL
LIN {X 0,Y 198.833,Z 665.791,A -85,B 0,C 180,E1 7575.109,E2 7575.109} C_VEL
LIN {X 0,Y 202.615,Z 649.923,A -85,B 0,C 180,E1 7573.857,E2 7573.857} C_VEL
LIN {X 0,Y 205.157,Z 633.141,A -85,B 0,C 180,E1 7573.004,E2 7573.004} C_VEL
LIN {X 0,Y 215.388,Z 522.939,A -85,B 0,C 180,E1 7569.686,E2 7569.686} C_VEL
LIN {X 0,Y 215.606,Z 495.453,A -85,B 0,C 180,E1 7567.546,E2 7567.546} C_VEL
LIN {X 0,Y 215.915,Z 490.055,A -85,B 0,C 180,E1 7567.05,E2 7567.05} C_VEL
LIN {X 0,Y 227.818,Z 446.411,A -85,B 0,C 180,E1 7561.761,E2 7561.761} C_VEL
LIN {X 0,Y 229.039,Z 441.918,A -85,B 0,C 180,E1 7561.189,E2 7561.189} C_VEL
LIN {X 0,Y 228.47,Z 434.651,A -85,B 0,C 180,E1 7557.995,E2 7557.995} C_VEL
LIN {X 0,Y 227.892,Z 428.743,A -85,B 0,C 180,E1 7554.462,E2 7554.462} C_VEL
LIN {X 0,Y 227.573,Z 424.262,A -85,B 0,C 180,E1 7550.645,E2 7550.645} C_VEL
LIN {X 0,Y 227.918,Z 421.264,A -85,B 0,C 180,E1 7546.039,E2 7546.039} C_VEL
LIN {X 0,Y 227.979,Z 421.154,A -85,B 0,C 180,E1 7544.659,E2 7544.659} C_VEL
LIN {X 0,Y 227.686,Z 422.083,A -85,B 0,C 180,E1 7543.82,E2 7543.82} C_VEL
LIN {X 0,Y 226.697,Z 425.422,A -85,B 0,C 180,E1 7542.879,E2 7542.879} C_VEL
LIN {X 0,Y 223.576,Z 435.876,A -85,B 0,C 180,E1 7541.116,E2 7541.116} C_VEL
LIN {X 0,Y 223.089,Z 438.023,A -85,B 0,C 180,E1 7540.503,E2 7540.503} C_VEL
LIN {X 0,Y 222.206,Z 443.371,A -85,B 0,C 180,E1 7538.626,E2 7538.626} C_VEL
LIN {X 0,Y 207.733,Z 490.679,A -85,B 0,C 180,E1 7535.62,E2 7535.62} C_VEL
LIN {X 0,Y 205.088,Z 506.601,A -85,B 0,C 180,E1 7534.872,E2 7534.872} C_VEL
LIN {X 0,Y 198.317,Z 572.607,A -85,B 0,C 180,E1 7532.448,E2 7532.448} C_VEL
LIN {X 0,Y 195.547,Z 601.102,A -85,B 0,C 180,E1 7531.377,E2 7531.377} C_VEL
LIN {X 0,Y 193.567,Z 624.291,A -85,B 0,C 180,E1 7530.326,E2 7530.326} C_VEL
LIN {X 0,Y 191.31,Z 647.465,A -85,B 0,C 180,E1 7529.182,E2 7529.182} C_VEL
LIN {X 0,Y 188.482,Z 663.492,A -85,B 0,C 180,E1 7527.963,E2 7527.963} C_VEL
LIN {X 0,Y 184.425,Z 679.041,A -85,B 0,C 180,E1 7526.318,E2 7526.318} C_VEL
LIN {X 0,Y 179.326,Z 693.956,A -85,B 0,C 180,E1 7524.22,E2 7524.22} C_VEL
LIN {X 0,Y 173.445,Z 707.897,A -85,B 0,C 180,E1 7521.621,E2 7521.621} C_VEL
LIN {X 0,Y 166.565,Z 721.606,A -85,B 0,C 180,E1 7518.219,E2 7518.219} C_VEL
LIN {X 0,Y 159.981,Z 733.088,A -85,B 0,C 180,E1 7514.42,E2 7514.42} C_VEL
LIN {X 0,Y 153.124,Z 743.911,A -85,B 0,C 180,E1 7509.602,E2 7509.602} C_VEL
LIN {X 0,Y 147.235,Z 752.62,A -85,B 0,C 180,E1 7504.303,E2 7504.303} C_VEL
LIN {X 0,Y 142.202,Z 759.961,A -85,B 0,C 180,E1 7498.1,E2 7498.1} C_VEL
LIN {X 0,Y 138.724,Z 765.29,A -85,B 0,C 180,E1 7491.562,E2 7491.562} C_VEL
LIN {X 0,Y 136.699,Z 768.974,A -85,B 0,C 180,E1 7484.395,E2 7484.395} C_VEL
